   1:L PR[91] 10mm/sec CNT100;
   1:  PR[GP1:91,1] = PR[GP1:90,1] + 6.355;
   1:  PR[GP1:91,2] = PR[GP1:90,2] + -5.589;
   1:L PR[91] 10mm/sec CNT100;
   1:  PR[GP1:91,1] = PR[GP1:90,1] + 7.372;
   1:  PR[GP1:91,2] = PR[GP1:90,2] + -9.674;
   1:L PR[91] 10mm/sec CNT100;
   1:  PR[GP1:91,1] = PR[GP1:90,1] + 8.367;
   1:  PR[GP1:91,2] = PR[GP1:90,2] + -12.675;
   1:L PR[91] 10mm/sec CNT100;
   1:  PR[GP1:91,1] = PR[GP1:90,1] + 10.321;
   1:  PR[GP1:91,2] = PR[GP1:90,2] + -16.925;
   1:L PR[91] 10mm/sec CNT100;
   1:  PR[GP1:91,1] = PR[GP1:90,1] + 13.045;
   1:  PR[GP1:91,2] = PR[GP1:90,2] + -20.757;
   1:L PR[91] 10mm/sec CNT100;
   1:  PR[GP1:91,1] = PR[GP1:90,1] + 14.879;
   1:  PR[GP1:91,2] = PR[GP1:90,2] + -23.159;
   1:L PR[91] 10mm/sec CNT100;
   1:  PR[GP1:91,1] = PR[GP1:90,1] + 18.319;
   1:  PR[GP1:91,2] = PR[GP1:90,2] + -26.468;
   1:L PR[91] 10mm/sec CNT100;
   1:  PR[GP1:91,1] = PR[GP1:90,1] + 22.355;
   1:  PR[GP1:91,2] = PR[GP1:90,2] + -29.107;
   1:L PR[91] 10mm/sec CNT100;
   1:  PR[GP1:91,1] = PR[GP1:90,1] + 24.727;
   1:  PR[GP1:91,2] = PR[GP1:90,2] + -30.680;
   1:L PR[91] 10mm/sec CNT100;
   1:  PR[GP1:91,1] = PR[GP1:90,1] + 29.246;
   1:  PR[GP1:91,2] = PR[GP1:90,2] + -32.548;
   1:L PR[91] 10mm/sec CNT100;
   1:  PR[GP1:91,1] = PR[GP1:90,1] + 34.105;
   1:  PR[GP1:91,2] = PR[GP1:90,2] + -33.559;
   1:L PR[91] 10mm/sec CNT100;
   1:  PR[GP1:91,1] = PR[GP1:90,1] + 36.667;
   1:  PR[GP1:91,2] = PR[GP1:90,2] + -34.223;
   1:L PR[91] 10mm/sec CNT100;
   1:  PR[GP1:91,1] = PR[GP1:90,1] + 41.699;
   1:  PR[GP1:91,2] = PR[GP1:90,2] + -34.315;
   1:L PR[91] 10mm/sec CNT100;
   1:  PR[GP1:91,1] = PR[GP1:90,1] + 44.031;
   1:  PR[GP1:91,2] = PR[GP1:90,2] + -34.139;
   1:L PR[91] 10mm/sec CNT100;
   1:  PR[GP1:91,1] = PR[GP1:90,1] + 49.115;
   1:  PR[GP1:91,2] = PR[GP1:90,2] + -33.273;
   1:L PR[91] 10mm/sec CNT100;
   1:  PR[GP1:91,1] = PR[GP1:90,1] + 53.961;
   1:  PR[GP1:91,2] = PR[GP1:90,2] + -31.473;
   1:L PR[91] 10mm/sec CNT100;
   1:  PR[GP1:91,1] = PR[GP1:90,1] + 55.965;
   1:  PR[GP1:91,2] = PR[GP1:90,2] + -30.610;
   1:L PR[91] 10mm/sec CNT100;
   1:  PR[GP1:91,1] = PR[GP1:90,1] + 60.444;
   1:  PR[GP1:91,2] = PR[GP1:90,2] + -27.909;
   1:L PR[91] 10mm/sec CNT100;
   1:  PR[GP1:91,1] = PR[GP1:90,1] + 64.372;
   1:  PR[GP1:91,2] = PR[GP1:90,2] + -24.396;
   1:L PR[91] 10mm/sec CNT100;
   1:  PR[GP1:91,1] = PR[GP1:90,1] + 65.892;
   1:  PR[GP1:91,2] = PR[GP1:90,2] + -23.011;
   1:L PR[91] 10mm/sec CNT100;
   1:  PR[GP1:91,1] = PR[GP1:90,1] + 69.105;
   1:  PR[GP1:91,2] = PR[GP1:90,2] + -18.822;
   1:L PR[91] 10mm/sec CNT100;
   1:  PR[GP1:91,1] = PR[GP1:90,1] + 71.512;
   1:  PR[GP1:91,2] = PR[GP1:90,2] + -14.052;
   1:L PR[91] 10mm/sec CNT100;
   1:  PR[GP1:91,1] = PR[GP1:90,1] + 72.452;
   1:  PR[GP1:91,2] = PR[GP1:90,2] + -12.328;
   1:L PR[91] 10mm/sec CNT100;
   1:  PR[GP1:91,1] = PR[GP1:90,1] + 73.920;
   1:  PR[GP1:91,2] = PR[GP1:90,2] + -7.231;
   1:L PR[91] 10mm/sec CNT100;
   1:  PR[GP1:91,1] = PR[GP1:90,1] + 74.423;
   1:  PR[GP1:91,2] = PR[GP1:90,2] + -1.863;
   1:L PR[91] 10mm/sec CNT100;
   1:  PR[GP1:91,1] = PR[GP1:90,1] + 74.736;
   1:  PR[GP1:91,2] = PR[GP1:90,2] + 0.017;
   1:L PR[91] 10mm/sec CNT100;
   1:  PR[GP1:91,1] = PR[GP1:90,1] + 74.236;
   1:  PR[GP1:91,2] = PR[GP1:90,2] + 5.360;
   1:L PR[91] 10mm/sec CNT100;
   1:  PR[GP1:91,1] = PR[GP1:90,1] + 73.926;
   1:  PR[GP1:91,2] = PR[GP1:90,2] + 7.201;
   1:L PR[91] 10mm/sec CNT100;
   1:  PR[GP1:91,1] = PR[GP1:90,1] + 72.449;
   1:  PR[GP1:91,2] = PR[GP1:90,2] + 12.328;
   1:L PR[91] 10mm/sec CNT100;
   1:  PR[GP1:91,1] = PR[GP1:90,1] + 70.034;
   1:  PR[GP1:91,2] = PR[GP1:90,2] + 17.114;
   1:L PR[91] 10mm/sec CNT100;
   1:  PR[GP1:91,1] = PR[GP1:90,1] + 69.111;
   1:  PR[GP1:91,2] = PR[GP1:90,2] + 18.805;
   1:L PR[91] 10mm/sec CNT100;
   1:  PR[GP1:91,1] = PR[GP1:90,1] + 65.893;
   1:  PR[GP1:91,2] = PR[GP1:90,2] + 23.000;
   1:L PR[91] 10mm/sec CNT100;
   1:  PR[GP1:91,1] = PR[GP1:90,1] + 61.915;
   1:  PR[GP1:91,2] = PR[GP1:90,2] + 26.557;
   1:L PR[91] 10mm/sec CNT100;
   1:  PR[GP1:91,1] = PR[GP1:90,1] + 60.442;
   1:  PR[GP1:91,2] = PR[GP1:90,2] + 27.901;
   1:L PR[91] 10mm/sec CNT100;
   1:  PR[GP1:91,1] = PR[GP1:90,1] + 55.978;
   1:  PR[GP1:91,2] = PR[GP1:90,2] + 30.593;
   1:L PR[91] 10mm/sec CNT100;
   1:  PR[GP1:91,1] = PR[GP1:90,1] + 51.021;
   1:  PR[GP1:91,2] = PR[GP1:90,2] + 32.434;
   1:L PR[91] 10mm/sec CNT100;
   1:  PR[GP1:91,1] = PR[GP1:90,1] + 49.099;
   1:  PR[GP1:91,2] = PR[GP1:90,2] + 33.267;
   1:L PR[91] 10mm/sec CNT100;
   1:  PR[GP1:91,1] = PR[GP1:90,1] + 44.031;
   1:  PR[GP1:91,2] = PR[GP1:90,2] + 34.130;
   1:L PR[91] 10mm/sec CNT100;
   1:  PR[GP1:91,1] = PR[GP1:90,1] + 41.699;
   1:  PR[GP1:91,2] = PR[GP1:90,2] + 34.306;
   1:L PR[91] 10mm/sec CNT100;
   1:  PR[GP1:91,1] = PR[GP1:90,1] + 36.653;
   1:  PR[GP1:91,2] = PR[GP1:90,2] + 34.214;
   1:L PR[91] 10mm/sec CNT100;
   1:  PR[GP1:91,1] = PR[GP1:90,1] + 31.699;
   1:  PR[GP1:91,2] = PR[GP1:90,2] + 33.183;
   1:L PR[91] 10mm/sec CNT100;
   1:  PR[GP1:91,1] = PR[GP1:90,1] + 29.260;
   1:  PR[GP1:91,2] = PR[GP1:90,2] + 32.545;
   1:L PR[91] 10mm/sec CNT100;
   1:  PR[GP1:91,1] = PR[GP1:90,1] + 24.725;
   1:  PR[GP1:91,2] = PR[GP1:90,2] + 30.670;
   1:L PR[91] 10mm/sec CNT100;
   1:  PR[GP1:91,1] = PR[GP1:90,1] + 20.585;
   1:  PR[GP1:91,2] = PR[GP1:90,2] + 27.963;
   1:L PR[91] 10mm/sec CNT100;
   1:  PR[GP1:91,1] = PR[GP1:90,1] + 18.321;
   1:  PR[GP1:91,2] = PR[GP1:90,2] + 26.461;
   1:L PR[91] 10mm/sec CNT100;
   1:  PR[GP1:91,1] = PR[GP1:90,1] + 14.886;
   1:  PR[GP1:91,2] = PR[GP1:90,2] + 23.157;
   1:L PR[91] 10mm/sec CNT100;
   1:  PR[GP1:91,1] = PR[GP1:90,1] + 12.088;
   1:  PR[GP1:91,2] = PR[GP1:90,2] + 19.220;
   1:L PR[91] 10mm/sec CNT100;
   1:  PR[GP1:91,1] = PR[GP1:90,1] + 10.317;
   1:  PR[GP1:91,2] = PR[GP1:90,2] + 16.907;
   1:L PR[91] 10mm/sec CNT100;
   1:  PR[GP1:91,1] = PR[GP1:90,1] + 8.367;
   1:  PR[GP1:91,2] = PR[GP1:90,2] + 12.666;
   1:L PR[91] 10mm/sec CNT100;
   1:  PR[GP1:91,1] = PR[GP1:90,1] + 7.372;
   1:  PR[GP1:91,2] = PR[GP1:90,2] + 9.665;
   1:L PR[91] 10mm/sec CNT100;
   1:  PR[GP1:91,1] = PR[GP1:90,1] + 6.354;
   1:  PR[GP1:91,2] = PR[GP1:90,2] + 5.577;
   1:L PR[91] 10mm/sec CNT100;
   1:  PR[GP1:91,1] = PR[GP1:90,1] + 6.524;
   1:  PR[GP1:91,2] = PR[GP1:90,2] + 5.479;
   1:L PR[91] 10mm/sec CNT100;
   1:  PR[GP1:91,1] = PR[GP1:90,1] + 5.914;
   1:  PR[GP1:91,2] = PR[GP1:90,2] + 4.305;
   1:L PR[91] 10mm/sec CNT100;
   1:  PR[GP1:91,1] = PR[GP1:90,1] + 4.686;
   1:  PR[GP1:91,2] = PR[GP1:90,2] + 2.087;
   1:L PR[91] 10mm/sec CNT100;
   1:  PR[GP1:91,1] = PR[GP1:90,1] + 4.389;
   1:  PR[GP1:91,2] = PR[GP1:90,2] + 1.764;
   1:L PR[91] 10mm/sec CNT100;
   1:  PR[GP1:91,1] = PR[GP1:90,1] + 3.955;
   1:  PR[GP1:91,2] = PR[GP1:90,2] + 1.465;
   1:L PR[91] 10mm/sec CNT100;
   1:  PR[GP1:91,1] = PR[GP1:90,1] + 1.605;
   1:  PR[GP1:91,2] = PR[GP1:90,2] + 0.594;
   1:L PR[91] 10mm/sec CNT100;
   1:  PR[GP1:91,1] = PR[GP1:90,1] + 0.862;
   1:  PR[GP1:91,2] = PR[GP1:90,2] + 0.396;
   1:L PR[91] 10mm/sec CNT100;
   1:  PR[GP1:91,1] = PR[GP1:90,1] + -0.072;
   1:L PR[91] 10mm/sec CNT100;
   1:  PR[GP1:91,1] = PR[GP1:90,1] + -1.424;
   1:  PR[GP1:91,2] = PR[GP1:90,2] + 0.956;
   1:  PR[GP1:91,3] = PR[GP1:90,3] + 11.970;
   1:L PR[91] 10mm/sec CNT100;
   1:  PR[GP1:91,1] = PR[GP1:90,1] + -1.547;
   1:  PR[GP1:91,2] = PR[GP1:90,2] + 0.962;
   1:L PR[91] 10mm/sec CNT100;
   1:  PR[GP1:91,1] = PR[GP1:90,1] + -3.479;
   1:  PR[GP1:91,2] = PR[GP1:90,2] + 1.726;
   1:L PR[91] 10mm/sec CNT100;
   1:  PR[GP1:91,1] = PR[GP1:90,1] + -4.374;
   1:  PR[GP1:91,2] = PR[GP1:90,2] + 3.341;
   1:L PR[91] 10mm/sec CNT100;
   1:  PR[GP1:91,1] = PR[GP1:90,1] + -4.406;
   1:  PR[GP1:91,2] = PR[GP1:90,2] + 3.371;
   1:L PR[91] 10mm/sec CNT100;
   1:  PR[GP1:91,1] = PR[GP1:90,1] + -5.693;
   1:  PR[GP1:91,2] = PR[GP1:90,2] + 5.463;
   1:L PR[91] 10mm/sec CNT100;
   1:  PR[GP1:91,1] = PR[GP1:90,1] + -5.438;
   1:  PR[GP1:91,2] = PR[GP1:90,2] + 5.607;
   1:L PR[91] 10mm/sec CNT100;
   1:  PR[GP1:91,1] = PR[GP1:90,1] + -6.155;
   1:  PR[GP1:91,2] = PR[GP1:90,2] + 8.483;
   1:L PR[91] 10mm/sec CNT100;
   1:  PR[GP1:91,1] = PR[GP1:90,1] + -7.832;
   1:  PR[GP1:91,2] = PR[GP1:90,2] + 13.544;
   1:L PR[91] 10mm/sec CNT100;
   1:  PR[GP1:91,1] = PR[GP1:90,1] + -9.289;
   1:  PR[GP1:91,2] = PR[GP1:90,2] + 16.715;
   1:L PR[91] 10mm/sec CNT100;
   1:  PR[GP1:91,1] = PR[GP1:90,1] + -11.324;
   1:  PR[GP1:91,2] = PR[GP1:90,2] + 19.577;
   1:L PR[91] 10mm/sec CNT100;
   1:  PR[GP1:91,1] = PR[GP1:90,1] + -14.416;
   1:  PR[GP1:91,2] = PR[GP1:90,2] + 23.625;
   1:L PR[91] 10mm/sec CNT100;
   1:  PR[GP1:91,1] = PR[GP1:90,1] + -17.052;
   1:  PR[GP1:91,2] = PR[GP1:90,2] + 26.160;
   1:L PR[91] 10mm/sec CNT100;
   1:  PR[GP1:91,1] = PR[GP1:90,1] + -20.154;
   1:  PR[GP1:91,2] = PR[GP1:90,2] + 28.188;
   1:L PR[91] 10mm/sec CNT100;
   1:  PR[GP1:91,1] = PR[GP1:90,1] + -24.154;
   1:  PR[GP1:91,2] = PR[GP1:90,2] + 30.842;
   1:L PR[91] 10mm/sec CNT100;
   1:  PR[GP1:91,1] = PR[GP1:90,1] + -27.722;
   1:  PR[GP1:91,2] = PR[GP1:90,2] + 32.317;
   1:L PR[91] 10mm/sec CNT100;
   1:  PR[GP1:91,1] = PR[GP1:90,1] + -31.573;
   1:  PR[GP1:91,2] = PR[GP1:90,2] + 33.118;
   1:L PR[91] 10mm/sec CNT100;
   1:  PR[GP1:91,1] = PR[GP1:90,1] + -35.898;
   1:  PR[GP1:91,2] = PR[GP1:90,2] + 34.238;
   1:L PR[91] 10mm/sec CNT100;
   1:  PR[GP1:91,1] = PR[GP1:90,1] + -39.986;
   1:  PR[GP1:91,2] = PR[GP1:90,2] + 34.312;
   1:L PR[91] 10mm/sec CNT100;
   1:  PR[GP1:91,1] = PR[GP1:90,1] + -43.926;
   1:  PR[GP1:91,2] = PR[GP1:90,2] + 34.016;
   1:L PR[91] 10mm/sec CNT100;
   1:  PR[GP1:91,1] = PR[GP1:90,1] + -48.152;
   1:  PR[GP1:91,2] = PR[GP1:90,2] + 33.296;
   1:L PR[91] 10mm/sec CNT100;
   1:  PR[GP1:91,1] = PR[GP1:90,1] + -52.182;
   1:  PR[GP1:91,2] = PR[GP1:90,2] + 31.799;
   1:L PR[91] 10mm/sec CNT100;
   1:  PR[GP1:91,1] = PR[GP1:90,1] + -55.570;
   1:  PR[GP1:91,2] = PR[GP1:90,2] + 30.339;
   1:L PR[91] 10mm/sec CNT100;
   1:  PR[GP1:91,1] = PR[GP1:90,1] + -59.354;
   1:  PR[GP1:91,2] = PR[GP1:90,2] + 28.057;
   1:L PR[91] 10mm/sec CNT100;
   1:  PR[GP1:91,1] = PR[GP1:90,1] + -62.677;
   1:  PR[GP1:91,2] = PR[GP1:90,2] + 25.086;
   1:L PR[91] 10mm/sec CNT100;
   1:  PR[GP1:91,1] = PR[GP1:90,1] + -65.248;
   1:  PR[GP1:91,2] = PR[GP1:90,2] + 22.743;
   1:L PR[91] 10mm/sec CNT100;
   1:  PR[GP1:91,1] = PR[GP1:90,1] + -67.992;
   1:  PR[GP1:91,2] = PR[GP1:90,2] + 19.165;
   1:L PR[91] 10mm/sec CNT100;
   1:  PR[GP1:91,1] = PR[GP1:90,1] + -70.053;
   1:  PR[GP1:91,2] = PR[GP1:90,2] + 15.082;
   1:L PR[91] 10mm/sec CNT100;
   1:  PR[GP1:91,1] = PR[GP1:90,1] + -71.643;
   1:  PR[GP1:91,2] = PR[GP1:90,2] + 12.163;
   1:L PR[91] 10mm/sec CNT100;
   1:  PR[GP1:91,1] = PR[GP1:90,1] + -72.905;
   1:  PR[GP1:91,2] = PR[GP1:90,2] + 7.782;
   1:L PR[91] 10mm/sec CNT100;
   1:  PR[GP1:91,1] = PR[GP1:90,1] + -73.338;
   1:  PR[GP1:91,2] = PR[GP1:90,2] + 3.156;
   1:L PR[91] 10mm/sec CNT100;
   1:  PR[GP1:91,1] = PR[GP1:90,1] + -73.869;
   1:  PR[GP1:91,2] = PR[GP1:90,2] + -0.026;
   1:L PR[91] 10mm/sec CNT100;
   1:  PR[GP1:91,1] = PR[GP1:90,1] + -73.436;
   1:  PR[GP1:91,2] = PR[GP1:90,2] + -4.653;
   1:L PR[91] 10mm/sec CNT100;
   1:  PR[GP1:91,1] = PR[GP1:90,1] + -72.911;
   1:  PR[GP1:91,2] = PR[GP1:90,2] + -7.770;
   1:L PR[91] 10mm/sec CNT100;
   1:  PR[GP1:91,1] = PR[GP1:90,1] + -71.641;
   1:  PR[GP1:91,2] = PR[GP1:90,2] + -12.181;
   1:L PR[91] 10mm/sec CNT100;
   1:  PR[GP1:91,1] = PR[GP1:90,1] + -69.561;
   1:  PR[GP1:91,2] = PR[GP1:90,2] + -16.301;
   1:L PR[91] 10mm/sec CNT100;
   1:  PR[GP1:91,1] = PR[GP1:90,1] + -67.998;
   1:  PR[GP1:91,2] = PR[GP1:90,2] + -19.166;
   1:L PR[91] 10mm/sec CNT100;
   1:  PR[GP1:91,1] = PR[GP1:90,1] + -65.249;
   1:  PR[GP1:91,2] = PR[GP1:90,2] + -22.750;
   1:L PR[91] 10mm/sec CNT100;
   1:  PR[GP1:91,1] = PR[GP1:90,1] + -61.846;
   1:  PR[GP1:91,2] = PR[GP1:90,2] + -25.794;
   1:L PR[91] 10mm/sec CNT100;
   1:  PR[GP1:91,1] = PR[GP1:90,1] + -59.352;
   1:  PR[GP1:91,2] = PR[GP1:90,2] + -28.067;
   1:L PR[91] 10mm/sec CNT100;
   1:  PR[GP1:91,1] = PR[GP1:90,1] + -55.583;
   1:  PR[GP1:91,2] = PR[GP1:90,2] + -30.340;
   1:L PR[91] 10mm/sec CNT100;
   1:  PR[GP1:91,1] = PR[GP1:90,1] + -51.387;
   1:  PR[GP1:91,2] = PR[GP1:90,2] + -31.899;
   1:L PR[91] 10mm/sec CNT100;
   1:  PR[GP1:91,1] = PR[GP1:90,1] + -48.136;
   1:  PR[GP1:91,2] = PR[GP1:90,2] + -33.307;
   1:L PR[91] 10mm/sec CNT100;
   1:  PR[GP1:91,1] = PR[GP1:90,1] + -43.926;
   1:  PR[GP1:91,2] = PR[GP1:90,2] + -34.025;
   1:L PR[91] 10mm/sec CNT100;
   1:  PR[GP1:91,1] = PR[GP1:90,1] + -39.986;
   1:  PR[GP1:91,2] = PR[GP1:90,2] + -34.321;
   1:L PR[91] 10mm/sec CNT100;
   1:  PR[GP1:91,1] = PR[GP1:90,1] + -35.883;
   1:  PR[GP1:91,2] = PR[GP1:90,2] + -34.247;
   1:L PR[91] 10mm/sec CNT100;
   1:  PR[GP1:91,1] = PR[GP1:90,1] + -31.854;
   1:  PR[GP1:91,2] = PR[GP1:90,2] + -33.408;
   1:L PR[91] 10mm/sec CNT100;
   1:  PR[GP1:91,1] = PR[GP1:90,1] + -27.736;
   1:  PR[GP1:91,2] = PR[GP1:90,2] + -32.331;
   1:L PR[91] 10mm/sec CNT100;
   1:  PR[GP1:91,1] = PR[GP1:90,1] + -24.152;
   1:  PR[GP1:91,2] = PR[GP1:90,2] + -30.850;
   1:L PR[91] 10mm/sec CNT100;
   1:  PR[GP1:91,1] = PR[GP1:90,1] + -20.874;
   1:  PR[GP1:91,2] = PR[GP1:90,2] + -28.706;
   1:L PR[91] 10mm/sec CNT100;
   1:  PR[GP1:91,1] = PR[GP1:90,1] + -17.054;
   1:  PR[GP1:91,2] = PR[GP1:90,2] + -26.171;
   1:L PR[91] 10mm/sec CNT100;
   1:  PR[GP1:91,1] = PR[GP1:90,1] + -14.423;
   1:  PR[GP1:91,2] = PR[GP1:90,2] + -23.641;
   1:L PR[91] 10mm/sec CNT100;
   1:  PR[GP1:91,1] = PR[GP1:90,1] + -12.272;
   1:  PR[GP1:91,2] = PR[GP1:90,2] + -20.613;
   1:L PR[91] 10mm/sec CNT100;
   1:  PR[GP1:91,1] = PR[GP1:90,1] + -9.285;
   1:  PR[GP1:91,2] = PR[GP1:90,2] + -16.713;
   1:L PR[91] 10mm/sec CNT100;
   1:  PR[GP1:91,1] = PR[GP1:90,1] + -7.832;
   1:  PR[GP1:91,2] = PR[GP1:90,2] + -13.553;
   1:L PR[91] 10mm/sec CNT100;
   1:  PR[GP1:91,1] = PR[GP1:90,1] + -6.155;
   1:  PR[GP1:91,2] = PR[GP1:90,2] + -8.493;
   1:L PR[91] 10mm/sec CNT100;
   1:  PR[GP1:91,1] = PR[GP1:90,1] + -5.437;
   1:  PR[GP1:91,2] = PR[GP1:90,2] + -5.610;
   1:L PR[91] 10mm/sec CNT100;
   1:  PR[GP1:91,1] = PR[GP1:90,1] + -5.649;
   1:  PR[GP1:91,2] = PR[GP1:90,2] + -5.486;
   1:L PR[91] 10mm/sec CNT100;
   1:  PR[GP1:91,1] = PR[GP1:90,1] + -4.810;
   1:  PR[GP1:91,2] = PR[GP1:90,2] + -3.871;
   1:L PR[91] 10mm/sec CNT100;
   1:  PR[GP1:91,1] = PR[GP1:90,1] + -3.915;
   1:  PR[GP1:91,2] = PR[GP1:90,2] + -2.254;
   1:L PR[91] 10mm/sec CNT100;
   1:  PR[GP1:91,1] = PR[GP1:90,1] + -3.482;
   1:  PR[GP1:91,2] = PR[GP1:90,2] + -1.784;
   1:L PR[91] 10mm/sec CNT100;
   1:  PR[GP1:91,1] = PR[GP1:90,1] + -2.834;
   1:  PR[GP1:91,2] = PR[GP1:90,2] + -1.337;
   1:L PR[91] 10mm/sec CNT100;
   1:  PR[GP1:91,1] = PR[GP1:90,1] + -1.161;
   1:  PR[GP1:91,2] = PR[GP1:90,2] + -0.717;
   1:L PR[91] 10mm/sec CNT100;
   1:  PR[GP1:91,1] = PR[GP1:90,1] + -0.101;
   1:  PR[GP1:91,2] = PR[GP1:90,2] + -0.435;
   1:L PR[91] 10mm/sec CNT100;
   1:  PR[GP1:91,1] = PR[GP1:90,1] + 0.024;
   1:  PR[GP1:91,2] = PR[GP1:90,2] + -0.404;
   1:L PR[91] 10mm/sec CNT100;
   1:  PR[GP1:91,1] = PR[GP1:90,1] + 0.838;
   1:L PR[91] 10mm/sec CNT100;
   1:  PR[GP1:91,1] = PR[GP1:90,1] + 2.244;
   1:  PR[GP1:91,2] = PR[GP1:90,2] + -0.965;
   1:L PR[91] 10mm/sec CNT100;
   1:  PR[GP1:91,1] = PR[GP1:90,1] + 2.368;
   1:  PR[GP1:91,2] = PR[GP1:90,2] + -0.970;
   1:L PR[91] 10mm/sec CNT100;
   1:  PR[GP1:91,1] = PR[GP1:90,1] + 4.300;
   1:  PR[GP1:91,2] = PR[GP1:90,2] + -1.735;
   1:L PR[91] 10mm/sec CNT100;
   1:  PR[GP1:91,1] = PR[GP1:90,1] + 5.194;
   1:  PR[GP1:91,2] = PR[GP1:90,2] + -3.350;
   1:L PR[91] 10mm/sec CNT100;
   1:  PR[GP1:91,1] = PR[GP1:90,1] + 5.227;
   1:  PR[GP1:91,2] = PR[GP1:90,2] + -3.380;
   1:L PR[91] 10mm/sec CNT100;
   1:  PR[GP1:91,1] = PR[GP1:90,1] + 6.512;
   1:  PR[GP1:91,2] = PR[GP1:90,2] + -5.470;
   1:L PR[91] 10mm/sec CNT100;
   1:  PR[GP1:91,1] = PR[GP1:90,1] + 6.258;
   1:  PR[GP1:91,2] = PR[GP1:90,2] + -5.615;
   1:L PR[91] 10mm/sec CNT100;
   1:  PR[GP1:91,1] = PR[GP1:90,1] + 6.975;
   1:  PR[GP1:91,2] = PR[GP1:90,2] + -8.494;
   1:L PR[91] 10mm/sec CNT100;
   1:  PR[GP1:91,1] = PR[GP1:90,1] + 8.652;
   1:  PR[GP1:91,2] = PR[GP1:90,2] + -13.551;
   1:L PR[91] 10mm/sec CNT100;
   1:  PR[GP1:91,1] = PR[GP1:90,1] + 10.109;
   1:  PR[GP1:91,2] = PR[GP1:90,2] + -16.721;
   1:L PR[91] 10mm/sec CNT100;
   1:  PR[GP1:91,1] = PR[GP1:90,1] + 12.144;
   1:  PR[GP1:91,2] = PR[GP1:90,2] + -19.584;
   1:L PR[91] 10mm/sec CNT100;
   1:  PR[GP1:91,1] = PR[GP1:90,1] + 15.236;
   1:  PR[GP1:91,2] = PR[GP1:90,2] + -23.633;
   1:L PR[91] 10mm/sec CNT100;
   1:  PR[GP1:91,1] = PR[GP1:90,1] + 17.872;
   1:  PR[GP1:91,2] = PR[GP1:90,2] + -26.169;
   1:L PR[91] 10mm/sec CNT100;
   1:  PR[GP1:91,1] = PR[GP1:90,1] + 20.974;
   1:  PR[GP1:91,2] = PR[GP1:90,2] + -28.196;
   1:L PR[91] 10mm/sec CNT100;
   1:  PR[GP1:91,1] = PR[GP1:90,1] + 24.974;
   1:  PR[GP1:91,2] = PR[GP1:90,2] + -30.850;
   1:L PR[91] 10mm/sec CNT100;
   1:  PR[GP1:91,1] = PR[GP1:90,1] + 28.542;
   1:  PR[GP1:91,2] = PR[GP1:90,2] + -32.325;
   1:L PR[91] 10mm/sec CNT100;
   1:  PR[GP1:91,1] = PR[GP1:90,1] + 32.393;
   1:  PR[GP1:91,2] = PR[GP1:90,2] + -33.126;
   1:L PR[91] 10mm/sec CNT100;
   1:  PR[GP1:91,1] = PR[GP1:90,1] + 36.718;
   1:  PR[GP1:91,2] = PR[GP1:90,2] + -34.247;
   1:L PR[91] 10mm/sec CNT100;
   1:  PR[GP1:91,1] = PR[GP1:90,1] + 40.805;
   1:  PR[GP1:91,2] = PR[GP1:90,2] + -34.321;
   1:L PR[91] 10mm/sec CNT100;
   1:  PR[GP1:91,1] = PR[GP1:90,1] + 44.746;
   1:  PR[GP1:91,2] = PR[GP1:90,2] + -34.025;
   1:L PR[91] 10mm/sec CNT100;
   1:  PR[GP1:91,1] = PR[GP1:90,1] + 48.972;
   1:  PR[GP1:91,2] = PR[GP1:90,2] + -33.305;
   1:L PR[91] 10mm/sec CNT100;
   1:  PR[GP1:91,1] = PR[GP1:90,1] + 53.002;
   1:  PR[GP1:91,2] = PR[GP1:90,2] + -31.807;
   1:L PR[91] 10mm/sec CNT100;
   1:  PR[GP1:91,1] = PR[GP1:90,1] + 56.390;
   1:  PR[GP1:91,2] = PR[GP1:90,2] + -30.348;
   1:L PR[91] 10mm/sec CNT100;
   1:  PR[GP1:91,1] = PR[GP1:90,1] + 60.174;
   1:  PR[GP1:91,2] = PR[GP1:90,2] + -28.066;
   1:L PR[91] 10mm/sec CNT100;
   1:  PR[GP1:91,1] = PR[GP1:90,1] + 63.498;
   1:  PR[GP1:91,2] = PR[GP1:90,2] + -25.095;
   1:L PR[91] 10mm/sec CNT100;
   1:  PR[GP1:91,1] = PR[GP1:90,1] + 66.068;
   1:  PR[GP1:91,2] = PR[GP1:90,2] + -22.752;
   1:L PR[91] 10mm/sec CNT100;
   1:  PR[GP1:91,1] = PR[GP1:90,1] + 68.813;
   1:  PR[GP1:91,2] = PR[GP1:90,2] + -19.173;
   1:L PR[91] 10mm/sec CNT100;
   1:  PR[GP1:91,1] = PR[GP1:90,1] + 70.873;
   1:  PR[GP1:91,2] = PR[GP1:90,2] + -15.091;
   1:L PR[91] 10mm/sec CNT100;
   1:  PR[GP1:91,1] = PR[GP1:90,1] + 72.464;
   1:  PR[GP1:91,2] = PR[GP1:90,2] + -12.173;
   1:L PR[91] 10mm/sec CNT100;
   1:  PR[GP1:91,1] = PR[GP1:90,1] + 73.725;
   1:  PR[GP1:91,2] = PR[GP1:90,2] + -7.792;
   1:L PR[91] 10mm/sec CNT100;
   1:  PR[GP1:91,1] = PR[GP1:90,1] + 74.159;
   1:  PR[GP1:91,2] = PR[GP1:90,2] + -3.166;
   1:L PR[91] 10mm/sec CNT100;
   1:  PR[GP1:91,1] = PR[GP1:90,1] + 74.690;
   1:  PR[GP1:91,2] = PR[GP1:90,2] + 0.017;
   1:L PR[91] 10mm/sec CNT100;
   1:  PR[GP1:91,1] = PR[GP1:90,1] + 74.256;
   1:  PR[GP1:91,2] = PR[GP1:90,2] + 4.644;
   1:L PR[91] 10mm/sec CNT100;
   1:  PR[GP1:91,1] = PR[GP1:90,1] + 73.731;
   1:  PR[GP1:91,2] = PR[GP1:90,2] + 7.762;
   1:L PR[91] 10mm/sec CNT100;
   1:  PR[GP1:91,1] = PR[GP1:90,1] + 72.461;
   1:  PR[GP1:91,2] = PR[GP1:90,2] + 12.173;
   1:L PR[91] 10mm/sec CNT100;
   1:  PR[GP1:91,1] = PR[GP1:90,1] + 70.382;
   1:  PR[GP1:91,2] = PR[GP1:90,2] + 16.293;
   1:L PR[91] 10mm/sec CNT100;
   1:  PR[GP1:91,1] = PR[GP1:90,1] + 68.819;
   1:  PR[GP1:91,2] = PR[GP1:90,2] + 19.157;
   1:L PR[91] 10mm/sec CNT100;
   1:  PR[GP1:91,1] = PR[GP1:90,1] + 66.070;
   1:  PR[GP1:91,2] = PR[GP1:90,2] + 22.741;
   1:L PR[91] 10mm/sec CNT100;
   1:  PR[GP1:91,1] = PR[GP1:90,1] + 62.666;
   1:  PR[GP1:91,2] = PR[GP1:90,2] + 25.784;
   1:L PR[91] 10mm/sec CNT100;
   1:  PR[GP1:91,1] = PR[GP1:90,1] + 60.172;
   1:  PR[GP1:91,2] = PR[GP1:90,2] + 28.059;
   1:L PR[91] 10mm/sec CNT100;
   1:  PR[GP1:91,1] = PR[GP1:90,1] + 56.403;
   1:  PR[GP1:91,2] = PR[GP1:90,2] + 30.332;
   1:L PR[91] 10mm/sec CNT100;
   1:  PR[GP1:91,1] = PR[GP1:90,1] + 52.207;
   1:  PR[GP1:91,2] = PR[GP1:90,2] + 31.890;
   1:L PR[91] 10mm/sec CNT100;
   1:  PR[GP1:91,1] = PR[GP1:90,1] + 48.956;
   1:  PR[GP1:91,2] = PR[GP1:90,2] + 33.298;
   1:L PR[91] 10mm/sec CNT100;
   1:  PR[GP1:91,1] = PR[GP1:90,1] + 44.746;
   1:  PR[GP1:91,2] = PR[GP1:90,2] + 34.016;
   1:L PR[91] 10mm/sec CNT100;
   1:  PR[GP1:91,1] = PR[GP1:90,1] + 40.805;
   1:  PR[GP1:91,2] = PR[GP1:90,2] + 34.312;
   1:L PR[91] 10mm/sec CNT100;
   1:  PR[GP1:91,1] = PR[GP1:90,1] + 36.703;
   1:  PR[GP1:91,2] = PR[GP1:90,2] + 34.238;
   1:L PR[91] 10mm/sec CNT100;
   1:  PR[GP1:91,1] = PR[GP1:90,1] + 32.674;
   1:  PR[GP1:91,2] = PR[GP1:90,2] + 33.399;
   1:L PR[91] 10mm/sec CNT100;
   1:  PR[GP1:91,1] = PR[GP1:90,1] + 28.556;
   1:  PR[GP1:91,2] = PR[GP1:90,2] + 32.322;
   1:L PR[91] 10mm/sec CNT100;
   1:  PR[GP1:91,1] = PR[GP1:90,1] + 24.972;
   1:  PR[GP1:91,2] = PR[GP1:90,2] + 30.840;
   1:L PR[91] 10mm/sec CNT100;
   1:  PR[GP1:91,1] = PR[GP1:90,1] + 21.693;
   1:  PR[GP1:91,2] = PR[GP1:90,2] + 28.696;
   1:L PR[91] 10mm/sec CNT100;
   1:  PR[GP1:91,1] = PR[GP1:90,1] + 17.874;
   1:  PR[GP1:91,2] = PR[GP1:90,2] + 26.161;
   1:L PR[91] 10mm/sec CNT100;
   1:  PR[GP1:91,1] = PR[GP1:90,1] + 15.243;
   1:  PR[GP1:91,2] = PR[GP1:90,2] + 23.631;
   1:L PR[91] 10mm/sec CNT100;
   1:  PR[GP1:91,1] = PR[GP1:90,1] + 13.091;
   1:  PR[GP1:91,2] = PR[GP1:90,2] + 20.604;
   1:L PR[91] 10mm/sec CNT100;
   1:  PR[GP1:91,1] = PR[GP1:90,1] + 10.105;
   1:  PR[GP1:91,2] = PR[GP1:90,2] + 16.703;
   1:L PR[91] 10mm/sec CNT100;
   1:  PR[GP1:91,1] = PR[GP1:90,1] + 8.652;
   1:  PR[GP1:91,2] = PR[GP1:90,2] + 13.542;
   1:L PR[91] 10mm/sec CNT100;
   1:  PR[GP1:91,1] = PR[GP1:90,1] + 6.975;
   1:  PR[GP1:91,2] = PR[GP1:90,2] + 8.484;
   1:L PR[91] 10mm/sec CNT100;
   1:  PR[GP1:91,1] = PR[GP1:90,1] + 6.258;
   1:  PR[GP1:91,2] = PR[GP1:90,2] + 5.602;
   1:L PR[91] 10mm/sec CNT100;
   1:  PR[GP1:91,1] = PR[GP1:90,1] + 6.470;
   1:  PR[GP1:91,2] = PR[GP1:90,2] + 5.479;
   1:L PR[91] 10mm/sec CNT100;
   1:  PR[GP1:91,1] = PR[GP1:90,1] + 5.631;
   1:  PR[GP1:91,2] = PR[GP1:90,2] + 3.863;
   1:L PR[91] 10mm/sec CNT100;
   1:  PR[GP1:91,1] = PR[GP1:90,1] + 4.735;
   1:  PR[GP1:91,2] = PR[GP1:90,2] + 2.246;
   1:L PR[91] 10mm/sec CNT100;
   1:  PR[GP1:91,1] = PR[GP1:90,1] + 4.302;
   1:  PR[GP1:91,2] = PR[GP1:90,2] + 1.775;
   1:L PR[91] 10mm/sec CNT100;
   1:  PR[GP1:91,1] = PR[GP1:90,1] + 3.654;
   1:  PR[GP1:91,2] = PR[GP1:90,2] + 1.329;
   1:L PR[91] 10mm/sec CNT100;
   1:  PR[GP1:91,1] = PR[GP1:90,1] + 1.982;
   1:  PR[GP1:91,2] = PR[GP1:90,2] + 0.708;
   1:L PR[91] 10mm/sec CNT100;
   1:  PR[GP1:91,1] = PR[GP1:90,1] + 0.919;
   1:  PR[GP1:91,2] = PR[GP1:90,2] + 0.425;
   1:L PR[91] 10mm/sec CNT100;
   1:  PR[GP1:91,1] = PR[GP1:90,1] + 0.796;
   1:  PR[GP1:91,2] = PR[GP1:90,2] + 0.396;
   1:L PR[91] 10mm/sec CNT100;
   1:  PR[GP1:91,1] = PR[GP1:90,1] + -0.018;
   1:L PR[91] 10mm/sec CNT100;
   1:  PR[GP1:91,1] = PR[GP1:90,1] + -0.616;
   1:  PR[GP1:91,2] = PR[GP1:90,2] + 0.693;
   1:  PR[GP1:91,3] = PR[GP1:90,3] + 13.300;
   1:L PR[91] 10mm/sec CNT100;
   1:  PR[GP1:91,1] = PR[GP1:90,1] + -0.790;
   1:  PR[GP1:91,2] = PR[GP1:90,2] + 0.701;
   1:L PR[91] 10mm/sec CNT100;
   1:  PR[GP1:91,1] = PR[GP1:90,1] + -3.381;
   1:  PR[GP1:91,2] = PR[GP1:90,2] + 1.726;
   1:L PR[91] 10mm/sec CNT100;
   1:  PR[GP1:91,1] = PR[GP1:90,1] + -3.935;
   1:  PR[GP1:91,2] = PR[GP1:90,2] + 2.726;
   1:L PR[91] 10mm/sec CNT100;
   1:  PR[GP1:91,1] = PR[GP1:90,1] + -3.985;
   1:  PR[GP1:91,2] = PR[GP1:90,2] + 2.772;
   1:L PR[91] 10mm/sec CNT100;
   1:  PR[GP1:91,1] = PR[GP1:90,1] + -4.673;
   1:  PR[GP1:91,2] = PR[GP1:90,2] + 3.890;
   1:L PR[91] 10mm/sec CNT100;
   1:  PR[GP1:91,1] = PR[GP1:90,1] + -5.310;
   1:  PR[GP1:91,2] = PR[GP1:90,2] + 5.066;
   1:L PR[91] 10mm/sec CNT100;
   1:  PR[GP1:91,1] = PR[GP1:90,1] + -5.369;
   1:  PR[GP1:91,2] = PR[GP1:90,2] + 5.616;
   1:L PR[91] 10mm/sec CNT100;
   1:  PR[GP1:91,1] = PR[GP1:90,1] + -5.342;
   1:  PR[GP1:91,2] = PR[GP1:90,2] + 5.632;
   1:L PR[91] 10mm/sec CNT100;
   1:  PR[GP1:91,1] = PR[GP1:90,1] + -5.758;
   1:  PR[GP1:91,2] = PR[GP1:90,2] + 7.303;
   1:L PR[91] 10mm/sec CNT100;
   1:  PR[GP1:91,1] = PR[GP1:90,1] + -8.117;
   1:  PR[GP1:91,2] = PR[GP1:90,2] + 14.421;
   1:L PR[91] 10mm/sec CNT100;
   1:  PR[GP1:91,1] = PR[GP1:90,1] + -9.078;
   1:  PR[GP1:91,2] = PR[GP1:90,2] + 16.511;
   1:L PR[91] 10mm/sec CNT100;
   1:  PR[GP1:91,1] = PR[GP1:90,1] + -10.424;
   1:  PR[GP1:91,2] = PR[GP1:90,2] + 18.405;
   1:L PR[91] 10mm/sec CNT100;
   1:  PR[GP1:91,1] = PR[GP1:90,1] + -14.774;
   1:  PR[GP1:91,2] = PR[GP1:90,2] + 24.099;
   1:L PR[91] 10mm/sec CNT100;
   1:  PR[GP1:91,1] = PR[GP1:90,1] + -16.606;
   1:  PR[GP1:91,2] = PR[GP1:90,2] + 25.861;
   1:L PR[91] 10mm/sec CNT100;
   1:  PR[GP1:91,1] = PR[GP1:90,1] + -18.773;
   1:  PR[GP1:91,2] = PR[GP1:90,2] + 27.278;
   1:L PR[91] 10mm/sec CNT100;
   1:  PR[GP1:91,1] = PR[GP1:90,1] + -24.402;
   1:  PR[GP1:91,2] = PR[GP1:90,2] + 31.012;
   1:L PR[91] 10mm/sec CNT100;
   1:  PR[GP1:91,1] = PR[GP1:90,1] + -27.019;
   1:  PR[GP1:91,2] = PR[GP1:90,2] + 32.094;
   1:L PR[91] 10mm/sec CNT100;
   1:  PR[GP1:91,1] = PR[GP1:90,1] + -29.862;
   1:  PR[GP1:91,2] = PR[GP1:90,2] + 32.685;
   1:L PR[91] 10mm/sec CNT100;
   1:  PR[GP1:91,1] = PR[GP1:90,1] + -35.949;
   1:  PR[GP1:91,2] = PR[GP1:90,2] + 34.262;
   1:L PR[91] 10mm/sec CNT100;
   1:  PR[GP1:91,1] = PR[GP1:90,1] + -39.092;
   1:  PR[GP1:91,2] = PR[GP1:90,2] + 34.319;
   1:L PR[91] 10mm/sec CNT100;
   1:  PR[GP1:91,1] = PR[GP1:90,1] + -44.641;
   1:  PR[GP1:91,2] = PR[GP1:90,2] + 33.901;
   1:L PR[91] 10mm/sec CNT100;
   1:  PR[GP1:91,1] = PR[GP1:90,1] + -48.009;
   1:  PR[GP1:91,2] = PR[GP1:90,2] + 33.327;
   1:L PR[91] 10mm/sec CNT100;
   1:  PR[GP1:91,1] = PR[GP1:90,1] + -51.223;
   1:  PR[GP1:91,2] = PR[GP1:90,2] + 32.133;
   1:L PR[91] 10mm/sec CNT100;
   1:  PR[GP1:91,1] = PR[GP1:90,1] + -55.995;
   1:  PR[GP1:91,2] = PR[GP1:90,2] + 30.078;
   1:L PR[91] 10mm/sec CNT100;
   1:  PR[GP1:91,1] = PR[GP1:90,1] + -59.085;
   1:  PR[GP1:91,2] = PR[GP1:90,2] + 28.215;
   1:L PR[91] 10mm/sec CNT100;
   1:  PR[GP1:91,1] = PR[GP1:90,1] + -61.802;
   1:  PR[GP1:91,2] = PR[GP1:90,2] + 25.785;
   1:L PR[91] 10mm/sec CNT100;
   1:  PR[GP1:91,1] = PR[GP1:90,1] + -65.424;
   1:  PR[GP1:91,2] = PR[GP1:90,2] + 22.484;
   1:L PR[91] 10mm/sec CNT100;
   1:  PR[GP1:91,1] = PR[GP1:90,1] + -67.700;
   1:  PR[GP1:91,2] = PR[GP1:90,2] + 19.516;
   1:L PR[91] 10mm/sec CNT100;
   1:  PR[GP1:91,1] = PR[GP1:90,1] + -69.414;
   1:  PR[GP1:91,2] = PR[GP1:90,2] + 16.122;
   1:L PR[91] 10mm/sec CNT100;
   1:  PR[GP1:91,1] = PR[GP1:90,1] + -71.655;
   1:  PR[GP1:91,2] = PR[GP1:90,2] + 12.007;
   1:L PR[91] 10mm/sec CNT100;
   1:  PR[GP1:91,1] = PR[GP1:90,1] + -72.710;
   1:  PR[GP1:91,2] = PR[GP1:90,2] + 8.343;
   1:L PR[91] 10mm/sec CNT100;
   1:  PR[GP1:91,1] = PR[GP1:90,1] + -73.074;
   1:  PR[GP1:91,2] = PR[GP1:90,2] + 4.459;
   1:L PR[91] 10mm/sec CNT100;
   1:  PR[GP1:91,1] = PR[GP1:90,1] + -73.823;
   1:  PR[GP1:91,2] = PR[GP1:90,2] + -0.026;
   1:L PR[91] 10mm/sec CNT100;
   1:  PR[GP1:91,1] = PR[GP1:90,1] + -73.456;
   1:  PR[GP1:91,2] = PR[GP1:90,2] + -3.937;
   1:L PR[91] 10mm/sec CNT100;
   1:  PR[GP1:91,1] = PR[GP1:90,1] + -72.717;
   1:  PR[GP1:91,2] = PR[GP1:90,2] + -8.330;
   1:L PR[91] 10mm/sec CNT100;
   1:  PR[GP1:91,1] = PR[GP1:90,1] + -71.652;
   1:  PR[GP1:91,2] = PR[GP1:90,2] + -12.025;
   1:L PR[91] 10mm/sec CNT100;
   1:  PR[GP1:91,1] = PR[GP1:90,1] + -69.909;
   1:  PR[GP1:91,2] = PR[GP1:90,2] + -15.479;
   1:L PR[91] 10mm/sec CNT100;
   1:  PR[GP1:91,1] = PR[GP1:90,1] + -67.706;
   1:  PR[GP1:91,2] = PR[GP1:90,2] + -19.518;
   1:L PR[91] 10mm/sec CNT100;
   1:  PR[GP1:91,1] = PR[GP1:90,1] + -65.426;
   1:  PR[GP1:91,2] = PR[GP1:90,2] + -22.491;
   1:L PR[91] 10mm/sec CNT100;
   1:  PR[GP1:91,1] = PR[GP1:90,1] + -62.596;
   1:  PR[GP1:91,2] = PR[GP1:90,2] + -25.021;
   1:L PR[91] 10mm/sec CNT100;
   1:  PR[GP1:91,1] = PR[GP1:90,1] + -59.082;
   1:  PR[GP1:91,2] = PR[GP1:90,2] + -28.225;
   1:L PR[91] 10mm/sec CNT100;
   1:  PR[GP1:91,1] = PR[GP1:90,1] + -56.008;
   1:  PR[GP1:91,2] = PR[GP1:90,2] + -30.078;
   1:L PR[91] 10mm/sec CNT100;
   1:  PR[GP1:91,1] = PR[GP1:90,1] + -52.573;
   1:  PR[GP1:91,2] = PR[GP1:90,2] + -31.354;
   1:L PR[91] 10mm/sec CNT100;
   1:  PR[GP1:91,1] = PR[GP1:90,1] + -47.993;
   1:  PR[GP1:91,2] = PR[GP1:90,2] + -33.339;
   1:L PR[91] 10mm/sec CNT100;
   1:  PR[GP1:91,1] = PR[GP1:90,1] + -44.641;
   1:  PR[GP1:91,2] = PR[GP1:90,2] + -33.910;
   1:L PR[91] 10mm/sec CNT100;
   1:  PR[GP1:91,1] = PR[GP1:90,1] + -39.092;
   1:  PR[GP1:91,2] = PR[GP1:90,2] + -34.328;
   1:L PR[91] 10mm/sec CNT100;
   1:  PR[GP1:91,1] = PR[GP1:90,1] + -35.934;
   1:  PR[GP1:91,2] = PR[GP1:90,2] + -34.270;
   1:L PR[91] 10mm/sec CNT100;
   1:  PR[GP1:91,1] = PR[GP1:90,1] + -32.829;
   1:  PR[GP1:91,2] = PR[GP1:90,2] + -33.624;
   1:L PR[91] 10mm/sec CNT100;
   1:  PR[GP1:91,1] = PR[GP1:90,1] + -27.033;
   1:  PR[GP1:91,2] = PR[GP1:90,2] + -32.108;
   1:L PR[91] 10mm/sec CNT100;
   1:  PR[GP1:91,1] = PR[GP1:90,1] + -24.400;
   1:  PR[GP1:91,2] = PR[GP1:90,2] + -31.020;
   1:L PR[91] 10mm/sec CNT100;
   1:  PR[GP1:91,1] = PR[GP1:90,1] + -21.983;
   1:  PR[GP1:91,2] = PR[GP1:90,2] + -29.440;
   1:L PR[91] 10mm/sec CNT100;
   1:  PR[GP1:91,1] = PR[GP1:90,1] + -16.607;
   1:  PR[GP1:91,2] = PR[GP1:90,2] + -25.872;
   1:L PR[91] 10mm/sec CNT100;
   1:  PR[GP1:91,1] = PR[GP1:90,1] + -14.781;
   1:  PR[GP1:91,2] = PR[GP1:90,2] + -24.115;
   1:L PR[91] 10mm/sec CNT100;
   1:  PR[GP1:91,1] = PR[GP1:90,1] + -13.276;
   1:  PR[GP1:91,2] = PR[GP1:90,2] + -21.997;
   1:L PR[91] 10mm/sec CNT100;
   1:  PR[GP1:91,1] = PR[GP1:90,1] + -9.073;
   1:  PR[GP1:91,2] = PR[GP1:90,2] + -16.510;
   1:L PR[91] 10mm/sec CNT100;
   1:  PR[GP1:91,1] = PR[GP1:90,1] + -8.117;
   1:  PR[GP1:91,2] = PR[GP1:90,2] + -14.430;
   1:L PR[91] 10mm/sec CNT100;
   1:  PR[GP1:91,1] = PR[GP1:90,1] + -5.758;
   1:  PR[GP1:91,2] = PR[GP1:90,2] + -7.313;
   1:L PR[91] 10mm/sec CNT100;
   1:  PR[GP1:91,1] = PR[GP1:90,1] + -5.340;
   1:  PR[GP1:91,2] = PR[GP1:90,2] + -5.635;
   1:L PR[91] 10mm/sec CNT100;
   1:  PR[GP1:91,1] = PR[GP1:90,1] + -5.371;
   1:  PR[GP1:91,2] = PR[GP1:90,2] + -5.618;
   1:L PR[91] 10mm/sec CNT100;
   1:  PR[GP1:91,1] = PR[GP1:90,1] + -5.314;
   1:  PR[GP1:91,2] = PR[GP1:90,2] + -5.104;
   1:L PR[91] 10mm/sec CNT100;
   1:  PR[GP1:91,1] = PR[GP1:90,1] + -4.965;
   1:  PR[GP1:91,2] = PR[GP1:90,2] + -4.273;
   1:L PR[91] 10mm/sec CNT100;
   1:  PR[GP1:91,1] = PR[GP1:90,1] + -4.526;
   1:  PR[GP1:91,2] = PR[GP1:90,2] + -3.429;
   1:L PR[91] 10mm/sec CNT100;
   1:  PR[GP1:91,1] = PR[GP1:90,1] + -3.964;
   1:  PR[GP1:91,2] = PR[GP1:90,2] + -2.413;
   1:L PR[91] 10mm/sec CNT100;
   1:  PR[GP1:91,1] = PR[GP1:90,1] + -3.395;
   1:  PR[GP1:91,2] = PR[GP1:90,2] + -1.795;
   1:L PR[91] 10mm/sec CNT100;
   1:  PR[GP1:91,1] = PR[GP1:90,1] + -2.533;
   1:  PR[GP1:91,2] = PR[GP1:90,2] + -1.201;
   1:L PR[91] 10mm/sec CNT100;
   1:  PR[GP1:91,1] = PR[GP1:90,1] + -1.538;
   1:  PR[GP1:91,2] = PR[GP1:90,2] + -0.832;
   1:L PR[91] 10mm/sec CNT100;
   1:  PR[GP1:91,1] = PR[GP1:90,1] + -0.919;
   1:  PR[GP1:91,2] = PR[GP1:90,2] + -0.667;
   1:L PR[91] 10mm/sec CNT100;
   1:  PR[GP1:91,1] = PR[GP1:90,1] + 0.173;
   1:  PR[GP1:91,2] = PR[GP1:90,2] + -0.404;
   1:L PR[91] 10mm/sec CNT100;
   1:  PR[GP1:91,1] = PR[GP1:90,1] + 0.690;
   1:L PR[91] 10mm/sec CNT100;
   1:  PR[GP1:91,1] = PR[GP1:90,1] + 1.437;
   1:  PR[GP1:91,2] = PR[GP1:90,2] + -0.702;
   1:L PR[91] 10mm/sec CNT100;
   1:  PR[GP1:91,1] = PR[GP1:90,1] + 1.611;
   1:  PR[GP1:91,2] = PR[GP1:90,2] + -0.710;
   1:L PR[91] 10mm/sec CNT100;
   1:  PR[GP1:91,1] = PR[GP1:90,1] + 4.202;
   1:  PR[GP1:91,2] = PR[GP1:90,2] + -1.735;
   1:L PR[91] 10mm/sec CNT100;
   1:  PR[GP1:91,1] = PR[GP1:90,1] + 4.756;
   1:  PR[GP1:91,2] = PR[GP1:90,2] + -2.736;
   1:L PR[91] 10mm/sec CNT100;
   1:  PR[GP1:91,1] = PR[GP1:90,1] + 4.806;
   1:  PR[GP1:91,2] = PR[GP1:90,2] + -2.781;
   1:L PR[91] 10mm/sec CNT100;
   1:  PR[GP1:91,1] = PR[GP1:90,1] + 5.494;
   1:  PR[GP1:91,2] = PR[GP1:90,2] + -3.900;
   1:L PR[91] 10mm/sec CNT100;
   1:  PR[GP1:91,1] = PR[GP1:90,1] + 6.130;
   1:  PR[GP1:91,2] = PR[GP1:90,2] + -5.075;
   1:L PR[91] 10mm/sec CNT100;
   1:  PR[GP1:91,1] = PR[GP1:90,1] + 6.190;
   1:  PR[GP1:91,2] = PR[GP1:90,2] + -5.625;
   1:L PR[91] 10mm/sec CNT100;
   1:  PR[GP1:91,1] = PR[GP1:90,1] + 6.162;
   1:  PR[GP1:91,2] = PR[GP1:90,2] + -5.640;
   1:L PR[91] 10mm/sec CNT100;
   1:  PR[GP1:91,1] = PR[GP1:90,1] + 6.578;
   1:  PR[GP1:91,2] = PR[GP1:90,2] + -7.314;
   1:L PR[91] 10mm/sec CNT100;
   1:  PR[GP1:91,1] = PR[GP1:90,1] + 8.936;
   1:  PR[GP1:91,2] = PR[GP1:90,2] + -14.427;
   1:L PR[91] 10mm/sec CNT100;
   1:  PR[GP1:91,1] = PR[GP1:90,1] + 9.897;
   1:  PR[GP1:91,2] = PR[GP1:90,2] + -16.517;
   1:L PR[91] 10mm/sec CNT100;
   1:  PR[GP1:91,1] = PR[GP1:90,1] + 11.243;
   1:  PR[GP1:91,2] = PR[GP1:90,2] + -18.411;
   1:L PR[91] 10mm/sec CNT100;
   1:  PR[GP1:91,1] = PR[GP1:90,1] + 15.593;
   1:  PR[GP1:91,2] = PR[GP1:90,2] + -24.107;
   1:L PR[91] 10mm/sec CNT100;
   1:  PR[GP1:91,1] = PR[GP1:90,1] + 17.425;
   1:  PR[GP1:91,2] = PR[GP1:90,2] + -25.869;
   1:L PR[91] 10mm/sec CNT100;
   1:  PR[GP1:91,1] = PR[GP1:90,1] + 19.593;
   1:  PR[GP1:91,2] = PR[GP1:90,2] + -27.286;
   1:L PR[91] 10mm/sec CNT100;
   1:  PR[GP1:91,1] = PR[GP1:90,1] + 25.221;
   1:  PR[GP1:91,2] = PR[GP1:90,2] + -31.020;
   1:L PR[91] 10mm/sec CNT100;
   1:  PR[GP1:91,1] = PR[GP1:90,1] + 27.838;
   1:  PR[GP1:91,2] = PR[GP1:90,2] + -32.102;
   1:L PR[91] 10mm/sec CNT100;
   1:  PR[GP1:91,1] = PR[GP1:90,1] + 30.681;
   1:  PR[GP1:91,2] = PR[GP1:90,2] + -32.694;
   1:L PR[91] 10mm/sec CNT100;
   1:  PR[GP1:91,1] = PR[GP1:90,1] + 36.769;
   1:  PR[GP1:91,2] = PR[GP1:90,2] + -34.270;
   1:L PR[91] 10mm/sec CNT100;
   1:  PR[GP1:91,1] = PR[GP1:90,1] + 39.912;
   1:  PR[GP1:91,2] = PR[GP1:90,2] + -34.328;
   1:L PR[91] 10mm/sec CNT100;
   1:  PR[GP1:91,1] = PR[GP1:90,1] + 45.461;
   1:  PR[GP1:91,2] = PR[GP1:90,2] + -33.910;
   1:L PR[91] 10mm/sec CNT100;
   1:  PR[GP1:91,1] = PR[GP1:90,1] + 48.829;
   1:  PR[GP1:91,2] = PR[GP1:90,2] + -33.336;
   1:L PR[91] 10mm/sec CNT100;
   1:  PR[GP1:91,1] = PR[GP1:90,1] + 52.043;
   1:  PR[GP1:91,2] = PR[GP1:90,2] + -32.142;
   1:L PR[91] 10mm/sec CNT100;
   1:  PR[GP1:91,1] = PR[GP1:90,1] + 56.816;
   1:  PR[GP1:91,2] = PR[GP1:90,2] + -30.087;
   1:L PR[91] 10mm/sec CNT100;
   1:  PR[GP1:91,1] = PR[GP1:90,1] + 59.905;
   1:  PR[GP1:91,2] = PR[GP1:90,2] + -28.224;
   1:L PR[91] 10mm/sec CNT100;
   1:  PR[GP1:91,1] = PR[GP1:90,1] + 62.623;
   1:  PR[GP1:91,2] = PR[GP1:90,2] + -25.794;
   1:L PR[91] 10mm/sec CNT100;
   1:  PR[GP1:91,1] = PR[GP1:90,1] + 66.245;
   1:  PR[GP1:91,2] = PR[GP1:90,2] + -22.492;
   1:L PR[91] 10mm/sec CNT100;
   1:  PR[GP1:91,1] = PR[GP1:90,1] + 68.521;
   1:  PR[GP1:91,2] = PR[GP1:90,2] + -19.525;
   1:L PR[91] 10mm/sec CNT100;
   1:  PR[GP1:91,1] = PR[GP1:90,1] + 70.234;
   1:  PR[GP1:91,2] = PR[GP1:90,2] + -16.130;
   1:L PR[91] 10mm/sec CNT100;
   1:  PR[GP1:91,1] = PR[GP1:90,1] + 72.476;
   1:  PR[GP1:91,2] = PR[GP1:90,2] + -12.018;
   1:L PR[91] 10mm/sec CNT100;
   1:  PR[GP1:91,1] = PR[GP1:90,1] + 73.531;
   1:  PR[GP1:91,2] = PR[GP1:90,2] + -8.354;
   1:L PR[91] 10mm/sec CNT100;
   1:  PR[GP1:91,1] = PR[GP1:90,1] + 73.895;
   1:  PR[GP1:91,2] = PR[GP1:90,2] + -4.470;
   1:L PR[91] 10mm/sec CNT100;
   1:  PR[GP1:91,1] = PR[GP1:90,1] + 74.643;
   1:  PR[GP1:91,2] = PR[GP1:90,2] + 0.017;
   1:L PR[91] 10mm/sec CNT100;
   1:  PR[GP1:91,1] = PR[GP1:90,1] + 74.277;
   1:  PR[GP1:91,2] = PR[GP1:90,2] + 3.928;
   1:L PR[91] 10mm/sec CNT100;
   1:  PR[GP1:91,1] = PR[GP1:90,1] + 73.537;
   1:  PR[GP1:91,2] = PR[GP1:90,2] + 8.323;
   1:L PR[91] 10mm/sec CNT100;
   1:  PR[GP1:91,1] = PR[GP1:90,1] + 72.473;
   1:  PR[GP1:91,2] = PR[GP1:90,2] + 12.018;
   1:L PR[91] 10mm/sec CNT100;
   1:  PR[GP1:91,1] = PR[GP1:90,1] + 70.730;
   1:  PR[GP1:91,2] = PR[GP1:90,2] + 15.472;
   1:L PR[91] 10mm/sec CNT100;
   1:  PR[GP1:91,1] = PR[GP1:90,1] + 68.527;
   1:  PR[GP1:91,2] = PR[GP1:90,2] + 19.508;
   1:L PR[91] 10mm/sec CNT100;
   1:  PR[GP1:91,1] = PR[GP1:90,1] + 66.247;
   1:  PR[GP1:91,2] = PR[GP1:90,2] + 22.481;
   1:L PR[91] 10mm/sec CNT100;
   1:  PR[GP1:91,1] = PR[GP1:90,1] + 63.417;
   1:  PR[GP1:91,2] = PR[GP1:90,2] + 25.011;
   1:L PR[91] 10mm/sec CNT100;
   1:  PR[GP1:91,1] = PR[GP1:90,1] + 59.902;
   1:  PR[GP1:91,2] = PR[GP1:90,2] + 28.217;
   1:L PR[91] 10mm/sec CNT100;
   1:  PR[GP1:91,1] = PR[GP1:90,1] + 56.829;
   1:  PR[GP1:91,2] = PR[GP1:90,2] + 30.070;
   1:L PR[91] 10mm/sec CNT100;
   1:  PR[GP1:91,1] = PR[GP1:90,1] + 53.394;
   1:  PR[GP1:91,2] = PR[GP1:90,2] + 31.346;
   1:L PR[91] 10mm/sec CNT100;
   1:  PR[GP1:91,1] = PR[GP1:90,1] + 48.813;
   1:  PR[GP1:91,2] = PR[GP1:90,2] + 33.330;
   1:L PR[91] 10mm/sec CNT100;
   1:  PR[GP1:91,1] = PR[GP1:90,1] + 45.461;
   1:  PR[GP1:91,2] = PR[GP1:90,2] + 33.901;
   1:L PR[91] 10mm/sec CNT100;
   1:  PR[GP1:91,1] = PR[GP1:90,1] + 39.912;
   1:  PR[GP1:91,2] = PR[GP1:90,2] + 34.319;
   1:L PR[91] 10mm/sec CNT100;
   1:  PR[GP1:91,1] = PR[GP1:90,1] + 36.754;
   1:  PR[GP1:91,2] = PR[GP1:90,2] + 34.261;
   1:L PR[91] 10mm/sec CNT100;
   1:  PR[GP1:91,1] = PR[GP1:90,1] + 33.649;
   1:  PR[GP1:91,2] = PR[GP1:90,2] + 33.615;
   1:L PR[91] 10mm/sec CNT100;
   1:  PR[GP1:91,1] = PR[GP1:90,1] + 27.852;
   1:  PR[GP1:91,2] = PR[GP1:90,2] + 32.099;
   1:L PR[91] 10mm/sec CNT100;
   1:  PR[GP1:91,1] = PR[GP1:90,1] + 25.219;
   1:  PR[GP1:91,2] = PR[GP1:90,2] + 31.010;
   1:L PR[91] 10mm/sec CNT100;
   1:  PR[GP1:91,1] = PR[GP1:90,1] + 22.802;
   1:  PR[GP1:91,2] = PR[GP1:90,2] + 29.430;
   1:L PR[91] 10mm/sec CNT100;
   1:  PR[GP1:91,1] = PR[GP1:90,1] + 17.427;
   1:  PR[GP1:91,2] = PR[GP1:90,2] + 25.862;
   1:L PR[91] 10mm/sec CNT100;
   1:  PR[GP1:91,1] = PR[GP1:90,1] + 15.600;
   1:  PR[GP1:91,2] = PR[GP1:90,2] + 24.105;
   1:L PR[91] 10mm/sec CNT100;
   1:  PR[GP1:91,1] = PR[GP1:90,1] + 14.095;
   1:  PR[GP1:91,2] = PR[GP1:90,2] + 21.988;
   1:L PR[91] 10mm/sec CNT100;
   1:  PR[GP1:91,1] = PR[GP1:90,1] + 9.893;
   1:  PR[GP1:91,2] = PR[GP1:90,2] + 16.499;
   1:L PR[91] 10mm/sec CNT100;
   1:  PR[GP1:91,1] = PR[GP1:90,1] + 8.936;
   1:  PR[GP1:91,2] = PR[GP1:90,2] + 14.418;
   1:L PR[91] 10mm/sec CNT100;
   1:  PR[GP1:91,1] = PR[GP1:90,1] + 6.578;
   1:  PR[GP1:91,2] = PR[GP1:90,2] + 7.303;
   1:L PR[91] 10mm/sec CNT100;
   1:  PR[GP1:91,1] = PR[GP1:90,1] + 6.161;
   1:  PR[GP1:91,2] = PR[GP1:90,2] + 5.628;
   1:L PR[91] 10mm/sec CNT100;
   1:  PR[GP1:91,1] = PR[GP1:90,1] + 6.191;
   1:  PR[GP1:91,2] = PR[GP1:90,2] + 5.610;
   1:L PR[91] 10mm/sec CNT100;
   1:  PR[GP1:91,1] = PR[GP1:90,1] + 6.135;
   1:  PR[GP1:91,2] = PR[GP1:90,2] + 5.096;
   1:L PR[91] 10mm/sec CNT100;
   1:  PR[GP1:91,1] = PR[GP1:90,1] + 5.787;
   1:  PR[GP1:91,2] = PR[GP1:90,2] + 4.267;
   1:L PR[91] 10mm/sec CNT100;
   1:  PR[GP1:91,1] = PR[GP1:90,1] + 5.347;
   1:  PR[GP1:91,2] = PR[GP1:90,2] + 3.420;
   1:L PR[91] 10mm/sec CNT100;
   1:  PR[GP1:91,1] = PR[GP1:90,1] + 4.785;
   1:  PR[GP1:91,2] = PR[GP1:90,2] + 2.405;
   1:L PR[91] 10mm/sec CNT100;
   1:  PR[GP1:91,1] = PR[GP1:90,1] + 4.215;
   1:  PR[GP1:91,2] = PR[GP1:90,2] + 1.786;
   1:L PR[91] 10mm/sec CNT100;
   1:  PR[GP1:91,1] = PR[GP1:90,1] + 3.354;
   1:  PR[GP1:91,2] = PR[GP1:90,2] + 1.192;
   1:L PR[91] 10mm/sec CNT100;
   1:  PR[GP1:91,1] = PR[GP1:90,1] + 2.358;
   1:  PR[GP1:91,2] = PR[GP1:90,2] + 0.823;
   1:L PR[91] 10mm/sec CNT100;
   1:  PR[GP1:91,1] = PR[GP1:90,1] + 1.738;
   1:  PR[GP1:91,2] = PR[GP1:90,2] + 0.658;
   1:L PR[91] 10mm/sec CNT100;
   1:  PR[GP1:91,1] = PR[GP1:90,1] + 0.647;
   1:  PR[GP1:91,2] = PR[GP1:90,2] + 0.396;
   1:L PR[91] 10mm/sec CNT100;
   1:  PR[GP1:91,1] = PR[GP1:90,1] + 0.130;
   1:L PR[91] 10mm/sec CNT100;
   1:  PR[GP1:91,1] = PR[GP1:90,1] + -0.033;
   1:  PR[GP1:91,2] = PR[GP1:90,2] + 0.440;
   1:  PR[GP1:91,3] = PR[GP1:90,3] + 14.630;
   1:L PR[91] 10mm/sec CNT100;
   1:  PR[GP1:91,1] = PR[GP1:90,1] + -3.284;
   1:  PR[GP1:91,2] = PR[GP1:90,2] + 1.727;
   1:L PR[91] 10mm/sec CNT100;
   1:  PR[GP1:91,1] = PR[GP1:90,1] + -3.497;
   1:  PR[GP1:91,2] = PR[GP1:90,2] + 2.112;
   1:L PR[91] 10mm/sec CNT100;
   1:  PR[GP1:91,1] = PR[GP1:90,1] + -3.564;
   1:  PR[GP1:91,2] = PR[GP1:90,2] + 2.173;
   1:L PR[91] 10mm/sec CNT100;
   1:  PR[GP1:91,1] = PR[GP1:90,1] + -3.820;
   1:  PR[GP1:91,2] = PR[GP1:90,2] + 2.589;
   1:L PR[91] 10mm/sec CNT100;
   1:  PR[GP1:91,1] = PR[GP1:90,1] + -5.162;
   1:  PR[GP1:91,2] = PR[GP1:90,2] + 5.067;
   1:L PR[91] 10mm/sec CNT100;
   1:  PR[GP1:91,1] = PR[GP1:90,1] + -5.211;
   1:  PR[GP1:91,2] = PR[GP1:90,2] + 5.520;
   1:L PR[91] 10mm/sec CNT100;
   1:  PR[GP1:91,1] = PR[GP1:90,1] + -5.361;
   1:  PR[GP1:91,2] = PR[GP1:90,2] + 6.122;
   1:L PR[91] 10mm/sec CNT100;
   1:  PR[GP1:91,1] = PR[GP1:90,1] + -8.402;
   1:  PR[GP1:91,2] = PR[GP1:90,2] + 15.298;
   1:L PR[91] 10mm/sec CNT100;
   1:  PR[GP1:91,1] = PR[GP1:90,1] + -8.866;
   1:  PR[GP1:91,2] = PR[GP1:90,2] + 16.308;
   1:L PR[91] 10mm/sec CNT100;
   1:  PR[GP1:91,1] = PR[GP1:90,1] + -9.523;
   1:  PR[GP1:91,2] = PR[GP1:90,2] + 17.232;
   1:L PR[91] 10mm/sec CNT100;
   1:  PR[GP1:91,1] = PR[GP1:90,1] + -15.131;
   1:  PR[GP1:91,2] = PR[GP1:90,2] + 24.573;
   1:L PR[91] 10mm/sec CNT100;
   1:  PR[GP1:91,1] = PR[GP1:90,1] + -16.160;
   1:  PR[GP1:91,2] = PR[GP1:90,2] + 25.563;
   1:L PR[91] 10mm/sec CNT100;
   1:  PR[GP1:91,1] = PR[GP1:90,1] + -24.649;
   1:  PR[GP1:91,2] = PR[GP1:90,2] + 31.182;
   1:L PR[91] 10mm/sec CNT100;
   1:  PR[GP1:91,1] = PR[GP1:90,1] + -26.315;
   1:  PR[GP1:91,2] = PR[GP1:90,2] + 31.871;
   1:L PR[91] 10mm/sec CNT100;
   1:  PR[GP1:91,1] = PR[GP1:90,1] + -28.151;
   1:  PR[GP1:91,2] = PR[GP1:90,2] + 32.253;
   1:L PR[91] 10mm/sec CNT100;
   1:  PR[GP1:91,1] = PR[GP1:90,1] + -36.000;
   1:  PR[GP1:91,2] = PR[GP1:90,2] + 34.285;
   1:L PR[91] 10mm/sec CNT100;
   1:  PR[GP1:91,1] = PR[GP1:90,1] + -38.199;
   1:  PR[GP1:91,2] = PR[GP1:90,2] + 34.325;
   1:L PR[91] 10mm/sec CNT100;
   1:  PR[GP1:91,1] = PR[GP1:90,1] + -45.356;
   1:  PR[GP1:91,2] = PR[GP1:90,2] + 33.787;
   1:L PR[91] 10mm/sec CNT100;
   1:  PR[GP1:91,1] = PR[GP1:90,1] + -47.866;
   1:  PR[GP1:91,2] = PR[GP1:90,2] + 33.359;
   1:L PR[91] 10mm/sec CNT100;
   1:  PR[GP1:91,1] = PR[GP1:90,1] + -50.265;
   1:  PR[GP1:91,2] = PR[GP1:90,2] + 32.468;
   1:L PR[91] 10mm/sec CNT100;
   1:  PR[GP1:91,1] = PR[GP1:90,1] + -56.421;
   1:  PR[GP1:91,2] = PR[GP1:90,2] + 29.816;
   1:L PR[91] 10mm/sec CNT100;
   1:  PR[GP1:91,1] = PR[GP1:90,1] + -58.815;
   1:  PR[GP1:91,2] = PR[GP1:90,2] + 28.372;
   1:L PR[91] 10mm/sec CNT100;
   1:  PR[GP1:91,1] = PR[GP1:90,1] + -60.928;
   1:  PR[GP1:91,2] = PR[GP1:90,2] + 26.483;
   1:L PR[91] 10mm/sec CNT100;
   1:  PR[GP1:91,1] = PR[GP1:90,1] + -65.601;
   1:  PR[GP1:91,2] = PR[GP1:90,2] + 22.225;
   1:L PR[91] 10mm/sec CNT100;
   1:  PR[GP1:91,1] = PR[GP1:90,1] + -67.408;
   1:  PR[GP1:91,2] = PR[GP1:90,2] + 19.868;
   1:L PR[91] 10mm/sec CNT100;
   1:  PR[GP1:91,1] = PR[GP1:90,1] + -68.775;
   1:  PR[GP1:91,2] = PR[GP1:90,2] + 17.161;
   1:L PR[91] 10mm/sec CNT100;
   1:  PR[GP1:91,1] = PR[GP1:90,1] + -71.667;
   1:  PR[GP1:91,2] = PR[GP1:90,2] + 11.851;
   1:L PR[91] 10mm/sec CNT100;
   1:  PR[GP1:91,1] = PR[GP1:90,1] + -72.516;
   1:  PR[GP1:91,2] = PR[GP1:90,2] + 8.904;
   1:L PR[91] 10mm/sec CNT100;
   1:  PR[GP1:91,1] = PR[GP1:90,1] + -72.811;
   1:  PR[GP1:91,2] = PR[GP1:90,2] + 5.762;
   1:L PR[91] 10mm/sec CNT100;
   1:  PR[GP1:91,1] = PR[GP1:90,1] + -73.776;
   1:  PR[GP1:91,2] = PR[GP1:90,2] + -0.026;
   1:L PR[91] 10mm/sec CNT100;
   1:  PR[GP1:91,1] = PR[GP1:90,1] + -73.477;
   1:  PR[GP1:91,2] = PR[GP1:90,2] + -3.221;
   1:L PR[91] 10mm/sec CNT100;
   1:  PR[GP1:91,1] = PR[GP1:90,1] + -72.522;
   1:  PR[GP1:91,2] = PR[GP1:90,2] + -8.891;
   1:L PR[91] 10mm/sec CNT100;
   1:  PR[GP1:91,1] = PR[GP1:90,1] + -71.664;
   1:  PR[GP1:91,2] = PR[GP1:90,2] + -11.869;
   1:L PR[91] 10mm/sec CNT100;
   1:  PR[GP1:91,1] = PR[GP1:90,1] + -70.257;
   1:  PR[GP1:91,2] = PR[GP1:90,2] + -14.658;
   1:L PR[91] 10mm/sec CNT100;
   1:  PR[GP1:91,1] = PR[GP1:90,1] + -67.414;
   1:  PR[GP1:91,2] = PR[GP1:90,2] + -19.869;
   1:L PR[91] 10mm/sec CNT100;
   1:  PR[GP1:91,1] = PR[GP1:90,1] + -65.603;
   1:  PR[GP1:91,2] = PR[GP1:90,2] + -22.231;
   1:L PR[91] 10mm/sec CNT100;
   1:  PR[GP1:91,1] = PR[GP1:90,1] + -63.347;
   1:  PR[GP1:91,2] = PR[GP1:90,2] + -24.248;
   1:L PR[91] 10mm/sec CNT100;
   1:  PR[GP1:91,1] = PR[GP1:90,1] + -58.813;
   1:  PR[GP1:91,2] = PR[GP1:90,2] + -28.382;
   1:L PR[91] 10mm/sec CNT100;
   1:  PR[GP1:91,1] = PR[GP1:90,1] + -56.434;
   1:  PR[GP1:91,2] = PR[GP1:90,2] + -29.817;
   1:L PR[91] 10mm/sec CNT100;
   1:  PR[GP1:91,1] = PR[GP1:90,1] + -53.760;
   1:  PR[GP1:91,2] = PR[GP1:90,2] + -30.810;
   1:L PR[91] 10mm/sec CNT100;
   1:  PR[GP1:91,1] = PR[GP1:90,1] + -47.850;
   1:  PR[GP1:91,2] = PR[GP1:90,2] + -33.371;
   1:L PR[91] 10mm/sec CNT100;
   1:  PR[GP1:91,1] = PR[GP1:90,1] + -45.356;
   1:  PR[GP1:91,2] = PR[GP1:90,2] + -33.796;
   1:L PR[91] 10mm/sec CNT100;
   1:  PR[GP1:91,1] = PR[GP1:90,1] + -38.199;
   1:  PR[GP1:91,2] = PR[GP1:90,2] + -34.334;
   1:L PR[91] 10mm/sec CNT100;
   1:  PR[GP1:91,1] = PR[GP1:90,1] + -35.985;
   1:  PR[GP1:91,2] = PR[GP1:90,2] + -34.294;
   1:L PR[91] 10mm/sec CNT100;
   1:  PR[GP1:91,1] = PR[GP1:90,1] + -33.805;
   1:  PR[GP1:91,2] = PR[GP1:90,2] + -33.840;
   1:L PR[91] 10mm/sec CNT100;
   1:  PR[GP1:91,1] = PR[GP1:90,1] + -26.329;
   1:  PR[GP1:91,2] = PR[GP1:90,2] + -31.886;
   1:L PR[91] 10mm/sec CNT100;
   1:  PR[GP1:91,1] = PR[GP1:90,1] + -24.648;
   1:  PR[GP1:91,2] = PR[GP1:90,2] + -31.190;
   1:L PR[91] 10mm/sec CNT100;
   1:  PR[GP1:91,1] = PR[GP1:90,1] + -23.092;
   1:  PR[GP1:91,2] = PR[GP1:90,2] + -30.174;
   1:L PR[91] 10mm/sec CNT100;
   1:  PR[GP1:91,1] = PR[GP1:90,1] + -16.160;
   1:  PR[GP1:91,2] = PR[GP1:90,2] + -25.572;
   1:L PR[91] 10mm/sec CNT100;
   1:  PR[GP1:91,1] = PR[GP1:90,1] + -15.139;
   1:  PR[GP1:91,2] = PR[GP1:90,2] + -24.589;
   1:L PR[91] 10mm/sec CNT100;
   1:  PR[GP1:91,1] = PR[GP1:90,1] + -14.280;
   1:  PR[GP1:91,2] = PR[GP1:90,2] + -23.381;
   1:L PR[91] 10mm/sec CNT100;
   1:  PR[GP1:91,1] = PR[GP1:90,1] + -8.862;
   1:  PR[GP1:91,2] = PR[GP1:90,2] + -16.307;
   1:L PR[91] 10mm/sec CNT100;
   1:  PR[GP1:91,1] = PR[GP1:90,1] + -8.402;
   1:  PR[GP1:91,2] = PR[GP1:90,2] + -15.307;
   1:L PR[91] 10mm/sec CNT100;
   1:  PR[GP1:91,1] = PR[GP1:90,1] + -5.361;
   1:  PR[GP1:91,2] = PR[GP1:90,2] + -6.133;
   1:L PR[91] 10mm/sec CNT100;
   1:  PR[GP1:91,1] = PR[GP1:90,1] + -5.213;
   1:  PR[GP1:91,2] = PR[GP1:90,2] + -5.537;
   1:L PR[91] 10mm/sec CNT100;
   1:  PR[GP1:91,1] = PR[GP1:90,1] + -5.166;
   1:  PR[GP1:91,2] = PR[GP1:90,2] + -5.106;
   1:L PR[91] 10mm/sec CNT100;
   1:  PR[GP1:91,1] = PR[GP1:90,1] + -4.410;
   1:  PR[GP1:91,2] = PR[GP1:90,2] + -3.308;
   1:L PR[91] 10mm/sec CNT100;
   1:  PR[GP1:91,1] = PR[GP1:90,1] + -4.016;
   1:  PR[GP1:91,2] = PR[GP1:90,2] + -2.575;
   1:L PR[91] 10mm/sec CNT100;
   1:  PR[GP1:91,1] = PR[GP1:90,1] + -3.308;
   1:  PR[GP1:91,2] = PR[GP1:90,2] + -1.805;
   1:L PR[91] 10mm/sec CNT100;
   1:  PR[GP1:91,1] = PR[GP1:90,1] + -2.223;
   1:  PR[GP1:91,2] = PR[GP1:90,2] + -1.058;
   1:L PR[91] 10mm/sec CNT100;
   1:  PR[GP1:91,1] = PR[GP1:90,1] + -1.754;
   1:  PR[GP1:91,2] = PR[GP1:90,2] + -0.903;
   1:L PR[91] 10mm/sec CNT100;
   1:  PR[GP1:91,1] = PR[GP1:90,1] + 0.403;
   1:  PR[GP1:91,2] = PR[GP1:90,2] + -0.385;
   1:L PR[91] 10mm/sec CNT100;
   1:  PR[GP1:91,1] = PR[GP1:90,1] + 0.596;
   1:  PR[GP1:91,2] = PR[GP1:90,2] + -0.438;
   1:L PR[91] 10mm/sec CNT100;
   1:  PR[GP1:91,1] = PR[GP1:90,1] + 0.854;
   1:  PR[GP1:91,2] = PR[GP1:90,2] + -0.449;
   1:L PR[91] 10mm/sec CNT100;
   1:  PR[GP1:91,1] = PR[GP1:90,1] + 4.104;
   1:  PR[GP1:91,2] = PR[GP1:90,2] + -1.736;
   1:L PR[91] 10mm/sec CNT100;
   1:  PR[GP1:91,1] = PR[GP1:90,1] + 4.317;
   1:  PR[GP1:91,2] = PR[GP1:90,2] + -2.121;
   1:L PR[91] 10mm/sec CNT100;
   1:  PR[GP1:91,1] = PR[GP1:90,1] + 4.385;
   1:  PR[GP1:91,2] = PR[GP1:90,2] + -2.182;
   1:L PR[91] 10mm/sec CNT100;
   1:  PR[GP1:91,1] = PR[GP1:90,1] + 4.641;
   1:  PR[GP1:91,2] = PR[GP1:90,2] + -2.599;
   1:L PR[91] 10mm/sec CNT100;
   1:  PR[GP1:91,1] = PR[GP1:90,1] + 5.982;
   1:  PR[GP1:91,2] = PR[GP1:90,2] + -5.077;
   1:L PR[91] 10mm/sec CNT100;
   1:  PR[GP1:91,1] = PR[GP1:90,1] + 6.032;
   1:  PR[GP1:91,2] = PR[GP1:90,2] + -5.531;
   1:L PR[91] 10mm/sec CNT100;
   1:  PR[GP1:91,1] = PR[GP1:90,1] + 6.182;
   1:  PR[GP1:91,2] = PR[GP1:90,2] + -6.133;
   1:L PR[91] 10mm/sec CNT100;
   1:  PR[GP1:91,1] = PR[GP1:90,1] + 9.221;
   1:  PR[GP1:91,2] = PR[GP1:90,2] + -15.303;
   1:L PR[91] 10mm/sec CNT100;
   1:  PR[GP1:91,1] = PR[GP1:90,1] + 9.686;
   1:  PR[GP1:91,2] = PR[GP1:90,2] + -16.313;
   1:L PR[91] 10mm/sec CNT100;
   1:  PR[GP1:91,1] = PR[GP1:90,1] + 10.343;
   1:  PR[GP1:91,2] = PR[GP1:90,2] + -17.237;
   1:L PR[91] 10mm/sec CNT100;
   1:  PR[GP1:91,1] = PR[GP1:90,1] + 15.950;
   1:  PR[GP1:91,2] = PR[GP1:90,2] + -24.581;
   1:L PR[91] 10mm/sec CNT100;
   1:  PR[GP1:91,1] = PR[GP1:90,1] + 16.979;
   1:  PR[GP1:91,2] = PR[GP1:90,2] + -25.571;
   1:L PR[91] 10mm/sec CNT100;
   1:  PR[GP1:91,1] = PR[GP1:90,1] + 25.468;
   1:  PR[GP1:91,2] = PR[GP1:90,2] + -31.190;
   1:L PR[91] 10mm/sec CNT100;
   1:  PR[GP1:91,1] = PR[GP1:90,1] + 27.134;
   1:  PR[GP1:91,2] = PR[GP1:90,2] + -31.879;
   1:L PR[91] 10mm/sec CNT100;
   1:  PR[GP1:91,1] = PR[GP1:90,1] + 28.969;
   1:  PR[GP1:91,2] = PR[GP1:90,2] + -32.261;
   1:L PR[91] 10mm/sec CNT100;
   1:  PR[GP1:91,1] = PR[GP1:90,1] + 36.819;
   1:  PR[GP1:91,2] = PR[GP1:90,2] + -34.294;
   1:L PR[91] 10mm/sec CNT100;
   1:  PR[GP1:91,1] = PR[GP1:90,1] + 39.018;
   1:  PR[GP1:91,2] = PR[GP1:90,2] + -34.334;
   1:L PR[91] 10mm/sec CNT100;
   1:  PR[GP1:91,1] = PR[GP1:90,1] + 46.175;
   1:  PR[GP1:91,2] = PR[GP1:90,2] + -33.796;
   1:L PR[91] 10mm/sec CNT100;
   1:  PR[GP1:91,1] = PR[GP1:90,1] + 48.686;
   1:  PR[GP1:91,2] = PR[GP1:90,2] + -33.368;
   1:L PR[91] 10mm/sec CNT100;
   1:  PR[GP1:91,1] = PR[GP1:90,1] + 51.085;
   1:  PR[GP1:91,2] = PR[GP1:90,2] + -32.477;
   1:L PR[91] 10mm/sec CNT100;
   1:  PR[GP1:91,1] = PR[GP1:90,1] + 57.241;
   1:  PR[GP1:91,2] = PR[GP1:90,2] + -29.826;
   1:L PR[91] 10mm/sec CNT100;
   1:  PR[GP1:91,1] = PR[GP1:90,1] + 59.635;
   1:  PR[GP1:91,2] = PR[GP1:90,2] + -28.382;
   1:L PR[91] 10mm/sec CNT100;
   1:  PR[GP1:91,1] = PR[GP1:90,1] + 61.748;
   1:  PR[GP1:91,2] = PR[GP1:90,2] + -26.493;
   1:L PR[91] 10mm/sec CNT100;
   1:  PR[GP1:91,1] = PR[GP1:90,1] + 66.421;
   1:  PR[GP1:91,2] = PR[GP1:90,2] + -22.233;
   1:L PR[91] 10mm/sec CNT100;
   1:  PR[GP1:91,1] = PR[GP1:90,1] + 68.229;
   1:  PR[GP1:91,2] = PR[GP1:90,2] + -19.876;
   1:L PR[91] 10mm/sec CNT100;
   1:  PR[GP1:91,1] = PR[GP1:90,1] + 69.595;
   1:  PR[GP1:91,2] = PR[GP1:90,2] + -17.169;
   1:L PR[91] 10mm/sec CNT100;
   1:  PR[GP1:91,1] = PR[GP1:90,1] + 72.488;
   1:  PR[GP1:91,2] = PR[GP1:90,2] + -11.863;
   1:L PR[91] 10mm/sec CNT100;
   1:  PR[GP1:91,1] = PR[GP1:90,1] + 73.337;
   1:  PR[GP1:91,2] = PR[GP1:90,2] + -8.915;
   1:L PR[91] 10mm/sec CNT100;
   1:  PR[GP1:91,1] = PR[GP1:90,1] + 73.631;
   1:  PR[GP1:91,2] = PR[GP1:90,2] + -5.774;
   1:L PR[91] 10mm/sec CNT100;
   1:  PR[GP1:91,1] = PR[GP1:90,1] + 74.597;
   1:  PR[GP1:91,2] = PR[GP1:90,2] + 0.017;
   1:L PR[91] 10mm/sec CNT100;
   1:  PR[GP1:91,1] = PR[GP1:90,1] + 74.297;
   1:  PR[GP1:91,2] = PR[GP1:90,2] + 3.213;
   1:L PR[91] 10mm/sec CNT100;
   1:  PR[GP1:91,1] = PR[GP1:90,1] + 73.343;
   1:  PR[GP1:91,2] = PR[GP1:90,2] + 8.885;
   1:L PR[91] 10mm/sec CNT100;
   1:  PR[GP1:91,1] = PR[GP1:90,1] + 72.485;
   1:  PR[GP1:91,2] = PR[GP1:90,2] + 11.863;
   1:L PR[91] 10mm/sec CNT100;
   1:  PR[GP1:91,1] = PR[GP1:90,1] + 71.078;
   1:  PR[GP1:91,2] = PR[GP1:90,2] + 14.652;
   1:L PR[91] 10mm/sec CNT100;
   1:  PR[GP1:91,1] = PR[GP1:90,1] + 68.235;
   1:  PR[GP1:91,2] = PR[GP1:90,2] + 19.860;
   1:L PR[91] 10mm/sec CNT100;
   1:  PR[GP1:91,1] = PR[GP1:90,1] + 66.423;
   1:  PR[GP1:91,2] = PR[GP1:90,2] + 22.221;
   1:L PR[91] 10mm/sec CNT100;
   1:  PR[GP1:91,1] = PR[GP1:90,1] + 64.167;
   1:  PR[GP1:91,2] = PR[GP1:90,2] + 24.238;
   1:L PR[91] 10mm/sec CNT100;
   1:  PR[GP1:91,1] = PR[GP1:90,1] + 59.633;
   1:  PR[GP1:91,2] = PR[GP1:90,2] + 28.375;
   1:L PR[91] 10mm/sec CNT100;
   1:  PR[GP1:91,1] = PR[GP1:90,1] + 57.254;
   1:  PR[GP1:91,2] = PR[GP1:90,2] + 29.809;
   1:L PR[91] 10mm/sec CNT100;
   1:  PR[GP1:91,1] = PR[GP1:90,1] + 54.580;
   1:  PR[GP1:91,2] = PR[GP1:90,2] + 30.802;
   1:L PR[91] 10mm/sec CNT100;
   1:  PR[GP1:91,1] = PR[GP1:90,1] + 48.670;
   1:  PR[GP1:91,2] = PR[GP1:90,2] + 33.362;
   1:L PR[91] 10mm/sec CNT100;
   1:  PR[GP1:91,1] = PR[GP1:90,1] + 46.175;
   1:  PR[GP1:91,2] = PR[GP1:90,2] + 33.787;
   1:L PR[91] 10mm/sec CNT100;
   1:  PR[GP1:91,1] = PR[GP1:90,1] + 39.018;
   1:  PR[GP1:91,2] = PR[GP1:90,2] + 34.325;
   1:L PR[91] 10mm/sec CNT100;
   1:  PR[GP1:91,1] = PR[GP1:90,1] + 36.804;
   1:  PR[GP1:91,2] = PR[GP1:90,2] + 34.285;
   1:L PR[91] 10mm/sec CNT100;
   1:  PR[GP1:91,1] = PR[GP1:90,1] + 34.624;
   1:  PR[GP1:91,2] = PR[GP1:90,2] + 33.831;
   1:L PR[91] 10mm/sec CNT100;
   1:  PR[GP1:91,1] = PR[GP1:90,1] + 27.148;
   1:  PR[GP1:91,2] = PR[GP1:90,2] + 31.876;
   1:L PR[91] 10mm/sec CNT100;
   1:  PR[GP1:91,1] = PR[GP1:90,1] + 25.467;
   1:  PR[GP1:91,2] = PR[GP1:90,2] + 31.181;
   1:L PR[91] 10mm/sec CNT100;
   1:  PR[GP1:91,1] = PR[GP1:90,1] + 23.911;
   1:  PR[GP1:91,2] = PR[GP1:90,2] + 30.164;
   1:L PR[91] 10mm/sec CNT100;
   1:  PR[GP1:91,1] = PR[GP1:90,1] + 16.979;
   1:  PR[GP1:91,2] = PR[GP1:90,2] + 25.562;
   1:L PR[91] 10mm/sec CNT100;
   1:  PR[GP1:91,1] = PR[GP1:90,1] + 15.958;
   1:  PR[GP1:91,2] = PR[GP1:90,2] + 24.580;
   1:L PR[91] 10mm/sec CNT100;
   1:  PR[GP1:91,1] = PR[GP1:90,1] + 15.099;
   1:  PR[GP1:91,2] = PR[GP1:90,2] + 23.371;
   1:L PR[91] 10mm/sec CNT100;
   1:  PR[GP1:91,1] = PR[GP1:90,1] + 9.681;
   1:  PR[GP1:91,2] = PR[GP1:90,2] + 16.294;
   1:L PR[91] 10mm/sec CNT100;
   1:  PR[GP1:91,1] = PR[GP1:90,1] + 9.221;
   1:  PR[GP1:91,2] = PR[GP1:90,2] + 15.295;
   1:L PR[91] 10mm/sec CNT100;
   1:  PR[GP1:91,1] = PR[GP1:90,1] + 6.181;
   1:  PR[GP1:91,2] = PR[GP1:90,2] + 6.122;
   1:L PR[91] 10mm/sec CNT100;
   1:  PR[GP1:91,1] = PR[GP1:90,1] + 6.033;
   1:  PR[GP1:91,2] = PR[GP1:90,2] + 5.528;
   1:L PR[91] 10mm/sec CNT100;
   1:  PR[GP1:91,1] = PR[GP1:90,1] + 5.986;
   1:  PR[GP1:91,2] = PR[GP1:90,2] + 5.098;
   1:L PR[91] 10mm/sec CNT100;
   1:  PR[GP1:91,1] = PR[GP1:90,1] + 5.232;
   1:  PR[GP1:91,2] = PR[GP1:90,2] + 3.301;
   1:L PR[91] 10mm/sec CNT100;
   1:  PR[GP1:91,1] = PR[GP1:90,1] + 4.837;
   1:  PR[GP1:91,2] = PR[GP1:90,2] + 2.567;
   1:L PR[91] 10mm/sec CNT100;
   1:  PR[GP1:91,1] = PR[GP1:90,1] + 4.128;
   1:  PR[GP1:91,2] = PR[GP1:90,2] + 1.797;
   1:L PR[91] 10mm/sec CNT100;
   1:  PR[GP1:91,1] = PR[GP1:90,1] + 3.044;
   1:  PR[GP1:91,2] = PR[GP1:90,2] + 1.049;
   1:L PR[91] 10mm/sec CNT100;
   1:  PR[GP1:91,1] = PR[GP1:90,1] + 2.573;
   1:  PR[GP1:91,2] = PR[GP1:90,2] + 0.894;
   1:L PR[91] 10mm/sec CNT100;
   1:  PR[GP1:91,1] = PR[GP1:90,1] + 0.347;
   1:  PR[GP1:91,2] = PR[GP1:90,2] + 0.368;
   1:L PR[91] 10mm/sec CNT100;
   1:  PR[GP1:91,1] = PR[GP1:90,1] + 0.191;
   1:  PR[GP1:91,2] = PR[GP1:90,2] + 0.430;
   1:L PR[91] 10mm/sec CNT100;
   1:  PR[GP1:91,1] = PR[GP1:90,1] + -2.902;
   1:  PR[GP1:91,2] = PR[GP1:90,2] + 1.855;
   1:  PR[GP1:91,3] = PR[GP1:90,3] + 15.960;
   1:L PR[91] 10mm/sec CNT100;
   1:  PR[GP1:91,1] = PR[GP1:90,1] + -3.131;
   1:  PR[GP1:91,2] = PR[GP1:90,2] + 2.042;
   1:L PR[91] 10mm/sec CNT100;
   1:  PR[GP1:91,1] = PR[GP1:90,1] + -5.016;
   1:  PR[GP1:91,2] = PR[GP1:90,2] + 5.352;
   1:L PR[91] 10mm/sec CNT100;
   1:  PR[GP1:91,1] = PR[GP1:90,1] + -8.669;
   1:  PR[GP1:91,2] = PR[GP1:90,2] + 16.121;
   1:L PR[91] 10mm/sec CNT100;
   1:  PR[GP1:91,1] = PR[GP1:90,1] + -15.489;
   1:  PR[GP1:91,2] = PR[GP1:90,2] + 25.048;
   1:L PR[91] 10mm/sec CNT100;
   1:  PR[GP1:91,1] = PR[GP1:90,1] + -15.713;
   1:  PR[GP1:91,2] = PR[GP1:90,2] + 25.264;
   1:L PR[91] 10mm/sec CNT100;
   1:  PR[GP1:91,1] = PR[GP1:90,1] + -24.897;
   1:  PR[GP1:91,2] = PR[GP1:90,2] + 31.353;
   1:L PR[91] 10mm/sec CNT100;
   1:  PR[GP1:91,1] = PR[GP1:90,1] + -25.611;
   1:  PR[GP1:91,2] = PR[GP1:90,2] + 31.648;
   1:L PR[91] 10mm/sec CNT100;
   1:  PR[GP1:91,1] = PR[GP1:90,1] + -26.439;
   1:  PR[GP1:91,2] = PR[GP1:90,2] + 31.820;
   1:L PR[91] 10mm/sec CNT100;
   1:  PR[GP1:91,1] = PR[GP1:90,1] + -36.051;
   1:  PR[GP1:91,2] = PR[GP1:90,2] + 34.309;
   1:L PR[91] 10mm/sec CNT100;
   1:  PR[GP1:91,1] = PR[GP1:90,1] + -37.306;
   1:  PR[GP1:91,2] = PR[GP1:90,2] + 34.332;
   1:L PR[91] 10mm/sec CNT100;
   1:  PR[GP1:91,1] = PR[GP1:90,1] + -46.070;
   1:  PR[GP1:91,2] = PR[GP1:90,2] + 33.672;
   1:L PR[91] 10mm/sec CNT100;
   1:  PR[GP1:91,1] = PR[GP1:90,1] + -47.723;
   1:  PR[GP1:91,2] = PR[GP1:90,2] + 33.391;
   1:L PR[91] 10mm/sec CNT100;
   1:  PR[GP1:91,1] = PR[GP1:90,1] + -49.306;
   1:  PR[GP1:91,2] = PR[GP1:90,2] + 32.802;
   1:L PR[91] 10mm/sec CNT100;
   1:  PR[GP1:91,1] = PR[GP1:90,1] + -56.846;
   1:  PR[GP1:91,2] = PR[GP1:90,2] + 29.554;
   1:L PR[91] 10mm/sec CNT100;
   1:  PR[GP1:91,1] = PR[GP1:90,1] + -58.546;
   1:  PR[GP1:91,2] = PR[GP1:90,2] + 28.530;
   1:L PR[91] 10mm/sec CNT100;
   1:  PR[GP1:91,1] = PR[GP1:90,1] + -60.053;
   1:  PR[GP1:91,2] = PR[GP1:90,2] + 27.182;
   1:L PR[91] 10mm/sec CNT100;
   1:  PR[GP1:91,1] = PR[GP1:90,1] + -65.778;
   1:  PR[GP1:91,2] = PR[GP1:90,2] + 21.965;
   1:L PR[91] 10mm/sec CNT100;
   1:  PR[GP1:91,1] = PR[GP1:90,1] + -67.116;
   1:  PR[GP1:91,2] = PR[GP1:90,2] + 20.220;
   1:L PR[91] 10mm/sec CNT100;
   1:  PR[GP1:91,1] = PR[GP1:90,1] + -68.136;
   1:  PR[GP1:91,2] = PR[GP1:90,2] + 18.200;
   1:L PR[91] 10mm/sec CNT100;
   1:  PR[GP1:91,1] = PR[GP1:90,1] + -71.679;
   1:  PR[GP1:91,2] = PR[GP1:90,2] + 11.696;
   1:L PR[91] 10mm/sec CNT100;
   1:  PR[GP1:91,1] = PR[GP1:90,1] + -72.322;
   1:  PR[GP1:91,2] = PR[GP1:90,2] + 9.464;
   1:L PR[91] 10mm/sec CNT100;
   1:  PR[GP1:91,1] = PR[GP1:90,1] + -72.547;
   1:  PR[GP1:91,2] = PR[GP1:90,2] + 7.065;
   1:L PR[91] 10mm/sec CNT100;
   1:  PR[GP1:91,1] = PR[GP1:90,1] + -73.730;
   1:  PR[GP1:91,2] = PR[GP1:90,2] + -0.026;
   1:L PR[91] 10mm/sec CNT100;
   1:  PR[GP1:91,1] = PR[GP1:90,1] + -73.497;
   1:  PR[GP1:91,2] = PR[GP1:90,2] + -2.506;
   1:L PR[91] 10mm/sec CNT100;
   1:  PR[GP1:91,1] = PR[GP1:90,1] + -72.328;
   1:  PR[GP1:91,2] = PR[GP1:90,2] + -9.452;
   1:L PR[91] 10mm/sec CNT100;
   1:  PR[GP1:91,1] = PR[GP1:90,1] + -71.676;
   1:  PR[GP1:91,2] = PR[GP1:90,2] + -11.714;
   1:L PR[91] 10mm/sec CNT100;
   1:  PR[GP1:91,1] = PR[GP1:90,1] + -70.605;
   1:  PR[GP1:91,2] = PR[GP1:90,2] + -13.837;
   1:L PR[91] 10mm/sec CNT100;
   1:  PR[GP1:91,1] = PR[GP1:90,1] + -67.122;
   1:  PR[GP1:91,2] = PR[GP1:90,2] + -20.221;
   1:L PR[91] 10mm/sec CNT100;
   1:  PR[GP1:91,1] = PR[GP1:90,1] + -65.780;
   1:  PR[GP1:91,2] = PR[GP1:90,2] + -21.972;
   1:L PR[91] 10mm/sec CNT100;
   1:  PR[GP1:91,1] = PR[GP1:90,1] + -64.098;
   1:  PR[GP1:91,2] = PR[GP1:90,2] + -23.475;
   1:L PR[91] 10mm/sec CNT100;
   1:  PR[GP1:91,1] = PR[GP1:90,1] + -58.543;
   1:  PR[GP1:91,2] = PR[GP1:90,2] + -28.540;
   1:L PR[91] 10mm/sec CNT100;
   1:  PR[GP1:91,1] = PR[GP1:90,1] + -56.860;
   1:  PR[GP1:91,2] = PR[GP1:90,2] + -29.555;
   1:L PR[91] 10mm/sec CNT100;
   1:  PR[GP1:91,1] = PR[GP1:90,1] + -54.946;
   1:  PR[GP1:91,2] = PR[GP1:90,2] + -30.266;
   1:L PR[91] 10mm/sec CNT100;
   1:  PR[GP1:91,1] = PR[GP1:90,1] + -47.707;
   1:  PR[GP1:91,2] = PR[GP1:90,2] + -33.402;
   1:L PR[91] 10mm/sec CNT100;
   1:  PR[GP1:91,1] = PR[GP1:90,1] + -46.070;
   1:  PR[GP1:91,2] = PR[GP1:90,2] + -33.681;
   1:L PR[91] 10mm/sec CNT100;
   1:  PR[GP1:91,1] = PR[GP1:90,1] + -37.306;
   1:  PR[GP1:91,2] = PR[GP1:90,2] + -34.341;
   1:L PR[91] 10mm/sec CNT100;
   1:  PR[GP1:91,1] = PR[GP1:90,1] + -36.036;
   1:  PR[GP1:91,2] = PR[GP1:90,2] + -34.318;
   1:L PR[91] 10mm/sec CNT100;
   1:  PR[GP1:91,1] = PR[GP1:90,1] + -34.780;
   1:  PR[GP1:91,2] = PR[GP1:90,2] + -34.056;
   1:L PR[91] 10mm/sec CNT100;
   1:  PR[GP1:91,1] = PR[GP1:90,1] + -25.625;
   1:  PR[GP1:91,2] = PR[GP1:90,2] + -31.663;
   1:L PR[91] 10mm/sec CNT100;
   1:  PR[GP1:91,1] = PR[GP1:90,1] + -24.897;
   1:  PR[GP1:91,2] = PR[GP1:90,2] + -31.361;
   1:L PR[91] 10mm/sec CNT100;
   1:  PR[GP1:91,1] = PR[GP1:90,1] + -15.713;
   1:  PR[GP1:91,2] = PR[GP1:90,2] + -25.273;
   1:L PR[91] 10mm/sec CNT100;
   1:  PR[GP1:91,1] = PR[GP1:90,1] + -15.496;
   1:  PR[GP1:91,2] = PR[GP1:90,2] + -25.064;
   1:L PR[91] 10mm/sec CNT100;
   1:  PR[GP1:91,1] = PR[GP1:90,1] + -15.284;
   1:  PR[GP1:91,2] = PR[GP1:90,2] + -24.765;
   1:L PR[91] 10mm/sec CNT100;
   1:  PR[GP1:91,1] = PR[GP1:90,1] + -8.669;
   1:  PR[GP1:91,2] = PR[GP1:90,2] + -16.129;
   1:L PR[91] 10mm/sec CNT100;
   1:  PR[GP1:91,1] = PR[GP1:90,1] + -5.033;
   1:  PR[GP1:91,2] = PR[GP1:90,2] + -5.411;
   1:L PR[91] 10mm/sec CNT100;
   1:  PR[GP1:91,1] = PR[GP1:90,1] + -4.722;
   1:  PR[GP1:91,2] = PR[GP1:90,2] + -4.538;
   1:L PR[91] 10mm/sec CNT100;
   1:  PR[GP1:91,1] = PR[GP1:90,1] + -4.045;
   1:  PR[GP1:91,2] = PR[GP1:90,2] + -2.946;
   1:L PR[91] 10mm/sec CNT100;
   1:  PR[GP1:91,1] = PR[GP1:90,1] + -3.559;
   1:  PR[GP1:91,2] = PR[GP1:90,2] + -2.518;
   1:L PR[91] 10mm/sec CNT100;
   1:  PR[GP1:91,1] = PR[GP1:90,1] + -2.954;
   1:  PR[GP1:91,2] = PR[GP1:90,2] + -1.894;
   1:L PR[91] 10mm/sec CNT100;
   1:  PR[GP1:91,1] = PR[GP1:90,1] + -1.938;
   1:  PR[GP1:91,2] = PR[GP1:90,2] + -1.389;
   1:L PR[91] 10mm/sec CNT100;
   1:  PR[GP1:91,1] = PR[GP1:90,1] + -1.147;
   1:  PR[GP1:91,2] = PR[GP1:90,2] + -0.940;
   1:L PR[91] 10mm/sec CNT100;
   1:  PR[GP1:91,1] = PR[GP1:90,1] + 0.073;
   1:  PR[GP1:91,2] = PR[GP1:90,2] + -0.669;
   1:L PR[91] 10mm/sec CNT100;
   1:  PR[GP1:91,1] = PR[GP1:90,1] + 0.335;
   1:  PR[GP1:91,2] = PR[GP1:90,2] + -0.667;
   1:L PR[91] 10mm/sec CNT100;
   1:  PR[GP1:91,1] = PR[GP1:90,1] + 3.723;
   1:  PR[GP1:91,2] = PR[GP1:90,2] + -1.864;
   1:L PR[91] 10mm/sec CNT100;
   1:  PR[GP1:91,1] = PR[GP1:90,1] + 3.952;
   1:  PR[GP1:91,2] = PR[GP1:90,2] + -2.052;
   1:L PR[91] 10mm/sec CNT100;
   1:  PR[GP1:91,1] = PR[GP1:90,1] + 5.324;
   1:  PR[GP1:91,2] = PR[GP1:90,2] + -4.467;
   1:L PR[91] 10mm/sec CNT100;
   1:  PR[GP1:91,1] = PR[GP1:90,1] + 5.682;
   1:  PR[GP1:91,2] = PR[GP1:90,2] + -5.148;
   1:L PR[91] 10mm/sec CNT100;
   1:  PR[GP1:91,1] = PR[GP1:90,1] + 5.818;
   1:  PR[GP1:91,2] = PR[GP1:90,2] + -5.308;
   1:L PR[91] 10mm/sec CNT100;
   1:  PR[GP1:91,1] = PR[GP1:90,1] + 9.489;
   1:  PR[GP1:91,2] = PR[GP1:90,2] + -16.125;
   1:L PR[91] 10mm/sec CNT100;
   1:  PR[GP1:91,1] = PR[GP1:90,1] + 16.307;
   1:  PR[GP1:91,2] = PR[GP1:90,2] + -25.056;
   1:L PR[91] 10mm/sec CNT100;
   1:  PR[GP1:91,1] = PR[GP1:90,1] + 16.532;
   1:  PR[GP1:91,2] = PR[GP1:90,2] + -25.272;
   1:L PR[91] 10mm/sec CNT100;
   1:  PR[GP1:91,1] = PR[GP1:90,1] + 25.716;
   1:  PR[GP1:91,2] = PR[GP1:90,2] + -31.360;
   1:L PR[91] 10mm/sec CNT100;
   1:  PR[GP1:91,1] = PR[GP1:90,1] + 26.430;
   1:  PR[GP1:91,2] = PR[GP1:90,2] + -31.656;
   1:L PR[91] 10mm/sec CNT100;
   1:  PR[GP1:91,1] = PR[GP1:90,1] + 27.258;
   1:  PR[GP1:91,2] = PR[GP1:90,2] + -31.828;
   1:L PR[91] 10mm/sec CNT100;
   1:  PR[GP1:91,1] = PR[GP1:90,1] + 36.870;
   1:  PR[GP1:91,2] = PR[GP1:90,2] + -34.318;
   1:L PR[91] 10mm/sec CNT100;
   1:  PR[GP1:91,1] = PR[GP1:90,1] + 38.125;
   1:  PR[GP1:91,2] = PR[GP1:90,2] + -34.341;
   1:L PR[91] 10mm/sec CNT100;
   1:  PR[GP1:91,1] = PR[GP1:90,1] + 46.890;
   1:  PR[GP1:91,2] = PR[GP1:90,2] + -33.681;
   1:L PR[91] 10mm/sec CNT100;
   1:  PR[GP1:91,1] = PR[GP1:90,1] + 48.543;
   1:  PR[GP1:91,2] = PR[GP1:90,2] + -33.400;
   1:L PR[91] 10mm/sec CNT100;
   1:  PR[GP1:91,1] = PR[GP1:90,1] + 50.126;
   1:  PR[GP1:91,2] = PR[GP1:90,2] + -32.811;
   1:L PR[91] 10mm/sec CNT100;
   1:  PR[GP1:91,1] = PR[GP1:90,1] + 57.666;
   1:  PR[GP1:91,2] = PR[GP1:90,2] + -29.564;
   1:L PR[91] 10mm/sec CNT100;
   1:  PR[GP1:91,1] = PR[GP1:90,1] + 59.366;
   1:  PR[GP1:91,2] = PR[GP1:90,2] + -28.540;
   1:L PR[91] 10mm/sec CNT100;
   1:  PR[GP1:91,1] = PR[GP1:90,1] + 60.873;
   1:  PR[GP1:91,2] = PR[GP1:90,2] + -27.191;
   1:L PR[91] 10mm/sec CNT100;
   1:  PR[GP1:91,1] = PR[GP1:90,1] + 66.598;
   1:  PR[GP1:91,2] = PR[GP1:90,2] + -21.973;
   1:L PR[91] 10mm/sec CNT100;
   1:  PR[GP1:91,1] = PR[GP1:90,1] + 67.937;
   1:  PR[GP1:91,2] = PR[GP1:90,2] + -20.228;
   1:L PR[91] 10mm/sec CNT100;
   1:  PR[GP1:91,1] = PR[GP1:90,1] + 68.956;
   1:  PR[GP1:91,2] = PR[GP1:90,2] + -18.208;
   1:L PR[91] 10mm/sec CNT100;
   1:  PR[GP1:91,1] = PR[GP1:90,1] + 72.500;
   1:  PR[GP1:91,2] = PR[GP1:90,2] + -11.708;
   1:L PR[91] 10mm/sec CNT100;
   1:  PR[GP1:91,1] = PR[GP1:90,1] + 73.142;
   1:  PR[GP1:91,2] = PR[GP1:90,2] + -9.476;
   1:L PR[91] 10mm/sec CNT100;
   1:  PR[GP1:91,1] = PR[GP1:90,1] + 73.367;
   1:  PR[GP1:91,2] = PR[GP1:90,2] + -7.077;
   1:L PR[91] 10mm/sec CNT100;
   1:  PR[GP1:91,1] = PR[GP1:90,1] + 74.550;
   1:  PR[GP1:91,2] = PR[GP1:90,2] + 0.017;
   1:L PR[91] 10mm/sec CNT100;
   1:  PR[GP1:91,1] = PR[GP1:90,1] + 74.318;
   1:  PR[GP1:91,2] = PR[GP1:90,2] + 2.497;
   1:L PR[91] 10mm/sec CNT100;
   1:  PR[GP1:91,1] = PR[GP1:90,1] + 73.148;
   1:  PR[GP1:91,2] = PR[GP1:90,2] + 9.446;
   1:L PR[91] 10mm/sec CNT100;
   1:  PR[GP1:91,1] = PR[GP1:90,1] + 72.497;
   1:  PR[GP1:91,2] = PR[GP1:90,2] + 11.708;
   1:L PR[91] 10mm/sec CNT100;
   1:  PR[GP1:91,1] = PR[GP1:90,1] + 71.426;
   1:  PR[GP1:91,2] = PR[GP1:90,2] + 13.831;
   1:L PR[91] 10mm/sec CNT100;
   1:  PR[GP1:91,1] = PR[GP1:90,1] + 67.943;
   1:  PR[GP1:91,2] = PR[GP1:90,2] + 20.211;
   1:L PR[91] 10mm/sec CNT100;
   1:  PR[GP1:91,1] = PR[GP1:90,1] + 66.600;
   1:  PR[GP1:91,2] = PR[GP1:90,2] + 21.962;
   1:L PR[91] 10mm/sec CNT100;
   1:  PR[GP1:91,1] = PR[GP1:90,1] + 64.918;
   1:  PR[GP1:91,2] = PR[GP1:90,2] + 23.465;
   1:L PR[91] 10mm/sec CNT100;
   1:  PR[GP1:91,1] = PR[GP1:90,1] + 59.363;
   1:  PR[GP1:91,2] = PR[GP1:90,2] + 28.532;
   1:L PR[91] 10mm/sec CNT100;
   1:  PR[GP1:91,1] = PR[GP1:90,1] + 57.680;
   1:  PR[GP1:91,2] = PR[GP1:90,2] + 29.547;
   1:L PR[91] 10mm/sec CNT100;
   1:  PR[GP1:91,1] = PR[GP1:90,1] + 55.766;
   1:  PR[GP1:91,2] = PR[GP1:90,2] + 30.258;
   1:L PR[91] 10mm/sec CNT100;
   1:  PR[GP1:91,1] = PR[GP1:90,1] + 48.527;
   1:  PR[GP1:91,2] = PR[GP1:90,2] + 33.393;
   1:L PR[91] 10mm/sec CNT100;
   1:  PR[GP1:91,1] = PR[GP1:90,1] + 46.890;
   1:  PR[GP1:91,2] = PR[GP1:90,2] + 33.672;
   1:L PR[91] 10mm/sec CNT100;
   1:  PR[GP1:91,1] = PR[GP1:90,1] + 38.125;
   1:  PR[GP1:91,2] = PR[GP1:90,2] + 34.332;
   1:L PR[91] 10mm/sec CNT100;
   1:  PR[GP1:91,1] = PR[GP1:90,1] + 36.855;
   1:  PR[GP1:91,2] = PR[GP1:90,2] + 34.309;
   1:L PR[91] 10mm/sec CNT100;
   1:  PR[GP1:91,1] = PR[GP1:90,1] + 35.599;
   1:  PR[GP1:91,2] = PR[GP1:90,2] + 34.047;
   1:L PR[91] 10mm/sec CNT100;
   1:  PR[GP1:91,1] = PR[GP1:90,1] + 26.444;
   1:  PR[GP1:91,2] = PR[GP1:90,2] + 31.653;
   1:L PR[91] 10mm/sec CNT100;
   1:  PR[GP1:91,1] = PR[GP1:90,1] + 25.716;
   1:  PR[GP1:91,2] = PR[GP1:90,2] + 31.351;
   1:L PR[91] 10mm/sec CNT100;
   1:  PR[GP1:91,1] = PR[GP1:90,1] + 16.532;
   1:  PR[GP1:91,2] = PR[GP1:90,2] + 25.263;
   1:L PR[91] 10mm/sec CNT100;
   1:  PR[GP1:91,1] = PR[GP1:90,1] + 16.315;
   1:  PR[GP1:91,2] = PR[GP1:90,2] + 25.054;
   1:L PR[91] 10mm/sec CNT100;
   1:  PR[GP1:91,1] = PR[GP1:90,1] + 16.103;
   1:  PR[GP1:91,2] = PR[GP1:90,2] + 24.755;
   1:L PR[91] 10mm/sec CNT100;
   1:  PR[GP1:91,1] = PR[GP1:90,1] + 9.488;
   1:  PR[GP1:91,2] = PR[GP1:90,2] + 16.116;
   1:L PR[91] 10mm/sec CNT100;
   1:  PR[GP1:91,1] = PR[GP1:90,1] + 5.853;
   1:  PR[GP1:91,2] = PR[GP1:90,2] + 5.403;
   1:L PR[91] 10mm/sec CNT100;
   1:  PR[GP1:91,1] = PR[GP1:90,1] + 5.542;
   1:  PR[GP1:91,2] = PR[GP1:90,2] + 4.531;
   1:L PR[91] 10mm/sec CNT100;
   1:  PR[GP1:91,1] = PR[GP1:90,1] + 4.866;
   1:  PR[GP1:91,2] = PR[GP1:90,2] + 2.937;
   1:L PR[91] 10mm/sec CNT100;
   1:  PR[GP1:91,1] = PR[GP1:90,1] + 4.380;
   1:  PR[GP1:91,2] = PR[GP1:90,2] + 2.509;
   1:L PR[91] 10mm/sec CNT100;
   1:  PR[GP1:91,1] = PR[GP1:90,1] + 3.774;
   1:  PR[GP1:91,2] = PR[GP1:90,2] + 1.885;
   1:L PR[91] 10mm/sec CNT100;
   1:  PR[GP1:91,1] = PR[GP1:90,1] + 2.759;
   1:  PR[GP1:91,2] = PR[GP1:90,2] + 1.380;
   1:L PR[91] 10mm/sec CNT100;
   1:  PR[GP1:91,1] = PR[GP1:90,1] + 1.967;
   1:  PR[GP1:91,2] = PR[GP1:90,2] + 0.931;
   1:L PR[91] 10mm/sec CNT100;
   1:  PR[GP1:91,1] = PR[GP1:90,1] + 0.748;
   1:  PR[GP1:91,2] = PR[GP1:90,2] + 0.660;
   1:L PR[91] 10mm/sec CNT100;
   1:  PR[GP1:91,1] = PR[GP1:90,1] + 0.486;
   1:  PR[GP1:91,2] = PR[GP1:90,2] + 0.658;
   1:L PR[91] 10mm/sec CNT100;
   1:  PR[GP1:91,1] = PR[GP1:90,1] + -0.489;
   1:  PR[GP1:91,2] = PR[GP1:90,2] + 1.445;
   1:  PR[GP1:91,3] = PR[GP1:90,3] + 17.290;
   1:L PR[91] 10mm/sec CNT100;
   1:  PR[GP1:91,1] = PR[GP1:90,1] + -0.834;
   1:  PR[GP1:91,2] = PR[GP1:90,2] + 1.594;
   1:L PR[91] 10mm/sec CNT100;
   1:  PR[GP1:91,1] = PR[GP1:90,1] + -2.634;
   1:  PR[GP1:91,2] = PR[GP1:90,2] + 2.244;
   1:L PR[91] 10mm/sec CNT100;
   1:  PR[GP1:91,1] = PR[GP1:90,1] + -4.963;
   1:  PR[GP1:91,2] = PR[GP1:90,2] + 6.311;
   1:L PR[91] 10mm/sec CNT100;
   1:  PR[GP1:91,1] = PR[GP1:90,1] + -7.913;
   1:  PR[GP1:91,2] = PR[GP1:90,2] + 15.001;
   1:L PR[91] 10mm/sec CNT100;
   1:  PR[GP1:91,1] = PR[GP1:90,1] + -8.812;
   1:  PR[GP1:91,2] = PR[GP1:90,2] + 16.799;
   1:L PR[91] 10mm/sec CNT100;
   1:  PR[GP1:91,1] = PR[GP1:90,1] + -14.903;
   1:  PR[GP1:91,2] = PR[GP1:90,2] + 24.619;
   1:L PR[91] 10mm/sec CNT100;
   1:  PR[GP1:91,1] = PR[GP1:90,1] + -15.727;
   1:  PR[GP1:91,2] = PR[GP1:90,2] + 25.445;
   1:L PR[91] 10mm/sec CNT100;
   1:  PR[GP1:91,1] = PR[GP1:90,1] + -24.933;
   1:  PR[GP1:91,2] = PR[GP1:90,2] + 31.423;
   1:L PR[91] 10mm/sec CNT100;
   1:  PR[GP1:91,1] = PR[GP1:90,1] + -25.079;
   1:  PR[GP1:91,2] = PR[GP1:90,2] + 31.498;
   1:L PR[91] 10mm/sec CNT100;
   1:  PR[GP1:91,1] = PR[GP1:90,1] + -27.678;
   1:  PR[GP1:91,2] = PR[GP1:90,2] + 32.151;
   1:L PR[91] 10mm/sec CNT100;
   1:  PR[GP1:91,1] = PR[GP1:90,1] + -36.102;
   1:  PR[GP1:91,2] = PR[GP1:90,2] + 34.333;
   1:L PR[91] 10mm/sec CNT100;
   1:  PR[GP1:91,1] = PR[GP1:90,1] + -36.413;
   1:  PR[GP1:91,2] = PR[GP1:90,2] + 34.338;
   1:L PR[91] 10mm/sec CNT100;
   1:  PR[GP1:91,1] = PR[GP1:90,1] + -46.785;
   1:  PR[GP1:91,2] = PR[GP1:90,2] + 33.558;
   1:L PR[91] 10mm/sec CNT100;
   1:  PR[GP1:91,1] = PR[GP1:90,1] + -47.580;
   1:  PR[GP1:91,2] = PR[GP1:90,2] + 33.422;
   1:L PR[91] 10mm/sec CNT100;
   1:  PR[GP1:91,1] = PR[GP1:90,1] + -48.348;
   1:  PR[GP1:91,2] = PR[GP1:90,2] + 33.137;
   1:L PR[91] 10mm/sec CNT100;
   1:  PR[GP1:91,1] = PR[GP1:90,1] + -57.272;
   1:  PR[GP1:91,2] = PR[GP1:90,2] + 29.293;
   1:L PR[91] 10mm/sec CNT100;
   1:  PR[GP1:91,1] = PR[GP1:90,1] + -58.276;
   1:  PR[GP1:91,2] = PR[GP1:90,2] + 28.687;
   1:L PR[91] 10mm/sec CNT100;
   1:  PR[GP1:91,1] = PR[GP1:90,1] + -59.179;
   1:  PR[GP1:91,2] = PR[GP1:90,2] + 27.880;
   1:L PR[91] 10mm/sec CNT100;
   1:  PR[GP1:91,1] = PR[GP1:90,1] + -65.955;
   1:  PR[GP1:91,2] = PR[GP1:90,2] + 21.706;
   1:L PR[91] 10mm/sec CNT100;
   1:  PR[GP1:91,1] = PR[GP1:90,1] + -66.824;
   1:  PR[GP1:91,2] = PR[GP1:90,2] + 20.572;
   1:L PR[91] 10mm/sec CNT100;
   1:  PR[GP1:91,1] = PR[GP1:90,1] + -67.497;
   1:  PR[GP1:91,2] = PR[GP1:90,2] + 19.239;
   1:L PR[91] 10mm/sec CNT100;
   1:  PR[GP1:91,1] = PR[GP1:90,1] + -71.691;
   1:  PR[GP1:91,2] = PR[GP1:90,2] + 11.540;
   1:L PR[91] 10mm/sec CNT100;
   1:  PR[GP1:91,1] = PR[GP1:90,1] + -72.127;
   1:  PR[GP1:91,2] = PR[GP1:90,2] + 10.025;
   1:L PR[91] 10mm/sec CNT100;
   1:  PR[GP1:91,1] = PR[GP1:90,1] + -72.283;
   1:  PR[GP1:91,2] = PR[GP1:90,2] + 8.368;
   1:L PR[91] 10mm/sec CNT100;
   1:  PR[GP1:91,1] = PR[GP1:90,1] + -73.683;
   1:  PR[GP1:91,2] = PR[GP1:90,2] + -0.026;
   1:L PR[91] 10mm/sec CNT100;
   1:  PR[GP1:91,1] = PR[GP1:90,1] + -73.518;
   1:  PR[GP1:91,2] = PR[GP1:90,2] + -1.790;
   1:L PR[91] 10mm/sec CNT100;
   1:  PR[GP1:91,1] = PR[GP1:90,1] + -72.133;
   1:  PR[GP1:91,2] = PR[GP1:90,2] + -10.013;
   1:L PR[91] 10mm/sec CNT100;
   1:  PR[GP1:91,1] = PR[GP1:90,1] + -71.688;
   1:  PR[GP1:91,2] = PR[GP1:90,2] + -11.558;
   1:L PR[91] 10mm/sec CNT100;
   1:  PR[GP1:91,1] = PR[GP1:90,1] + -70.953;
   1:  PR[GP1:91,2] = PR[GP1:90,2] + -13.016;
   1:L PR[91] 10mm/sec CNT100;
   1:  PR[GP1:91,1] = PR[GP1:90,1] + -66.830;
   1:  PR[GP1:91,2] = PR[GP1:90,2] + -20.573;
   1:L PR[91] 10mm/sec CNT100;
   1:  PR[GP1:91,1] = PR[GP1:90,1] + -65.956;
   1:  PR[GP1:91,2] = PR[GP1:90,2] + -21.712;
   1:L PR[91] 10mm/sec CNT100;
   1:  PR[GP1:91,1] = PR[GP1:90,1] + -64.849;
   1:  PR[GP1:91,2] = PR[GP1:90,2] + -22.703;
   1:L PR[91] 10mm/sec CNT100;
   1:  PR[GP1:91,1] = PR[GP1:90,1] + -58.274;
   1:  PR[GP1:91,2] = PR[GP1:90,2] + -28.697;
   1:L PR[91] 10mm/sec CNT100;
   1:  PR[GP1:91,1] = PR[GP1:90,1] + -57.285;
   1:  PR[GP1:91,2] = PR[GP1:90,2] + -29.294;
   1:L PR[91] 10mm/sec CNT100;
   1:  PR[GP1:91,1] = PR[GP1:90,1] + -56.133;
   1:  PR[GP1:91,2] = PR[GP1:90,2] + -29.722;
   1:L PR[91] 10mm/sec CNT100;
   1:  PR[GP1:91,1] = PR[GP1:90,1] + -47.564;
   1:  PR[GP1:91,2] = PR[GP1:90,2] + -33.434;
   1:L PR[91] 10mm/sec CNT100;
   1:  PR[GP1:91,1] = PR[GP1:90,1] + -46.785;
   1:  PR[GP1:91,2] = PR[GP1:90,2] + -33.567;
   1:L PR[91] 10mm/sec CNT100;
   1:  PR[GP1:91,1] = PR[GP1:90,1] + -36.413;
   1:  PR[GP1:91,2] = PR[GP1:90,2] + -34.347;
   1:L PR[91] 10mm/sec CNT100;
   1:  PR[GP1:91,1] = PR[GP1:90,1] + -36.087;
   1:  PR[GP1:91,2] = PR[GP1:90,2] + -34.341;
   1:L PR[91] 10mm/sec CNT100;
   1:  PR[GP1:91,1] = PR[GP1:90,1] + -35.755;
   1:  PR[GP1:91,2] = PR[GP1:90,2] + -34.272;
   1:L PR[91] 10mm/sec CNT100;
   1:  PR[GP1:91,1] = PR[GP1:90,1] + -27.679;
   1:  PR[GP1:91,2] = PR[GP1:90,2] + -32.160;
   1:L PR[91] 10mm/sec CNT100;
   1:  PR[GP1:91,1] = PR[GP1:90,1] + -25.079;
   1:  PR[GP1:91,2] = PR[GP1:90,2] + -31.507;
   1:L PR[91] 10mm/sec CNT100;
   1:  PR[GP1:91,1] = PR[GP1:90,1] + -24.933;
   1:  PR[GP1:91,2] = PR[GP1:90,2] + -31.432;
   1:L PR[91] 10mm/sec CNT100;
   1:  PR[GP1:91,1] = PR[GP1:90,1] + -15.727;
   1:  PR[GP1:91,2] = PR[GP1:90,2] + -25.454;
   1:L PR[91] 10mm/sec CNT100;
   1:  PR[GP1:91,1] = PR[GP1:90,1] + -14.903;
   1:  PR[GP1:91,2] = PR[GP1:90,2] + -24.628;
   1:L PR[91] 10mm/sec CNT100;
   1:  PR[GP1:91,1] = PR[GP1:90,1] + -8.812;
   1:  PR[GP1:91,2] = PR[GP1:90,2] + -16.808;
   1:L PR[91] 10mm/sec CNT100;
   1:  PR[GP1:91,1] = PR[GP1:90,1] + -7.914;
   1:  PR[GP1:91,2] = PR[GP1:90,2] + -15.014;
   1:L PR[91] 10mm/sec CNT100;
   1:  PR[GP1:91,1] = PR[GP1:90,1] + -4.980;
   1:  PR[GP1:91,2] = PR[GP1:90,2] + -6.371;
   1:L PR[91] 10mm/sec CNT100;
   1:  PR[GP1:91,1] = PR[GP1:90,1] + -4.084;
   1:  PR[GP1:91,2] = PR[GP1:90,2] + -3.857;
   1:L PR[91] 10mm/sec CNT100;
   1:  PR[GP1:91,1] = PR[GP1:90,1] + -3.238;
   1:  PR[GP1:91,2] = PR[GP1:90,2] + -2.922;
   1:L PR[91] 10mm/sec CNT100;
   1:  PR[GP1:91,1] = PR[GP1:90,1] + -2.608;
   1:  PR[GP1:91,2] = PR[GP1:90,2] + -2.367;
   1:L PR[91] 10mm/sec CNT100;
   1:  PR[GP1:91,1] = PR[GP1:90,1] + -2.371;
   1:  PR[GP1:91,2] = PR[GP1:90,2] + -2.122;
   1:L PR[91] 10mm/sec CNT100;
   1:  PR[GP1:91,1] = PR[GP1:90,1] + -1.937;
   1:  PR[GP1:91,2] = PR[GP1:90,2] + -1.948;
   1:L PR[91] 10mm/sec CNT100;
   1:  PR[GP1:91,1] = PR[GP1:90,1] + -0.652;
   1:  PR[GP1:91,2] = PR[GP1:90,2] + -1.293;
   1:L PR[91] 10mm/sec CNT100;
   1:  PR[GP1:91,1] = PR[GP1:90,1] + 1.309;
   1:  PR[GP1:91,2] = PR[GP1:90,2] + -1.454;
   1:L PR[91] 10mm/sec CNT100;
   1:  PR[GP1:91,1] = PR[GP1:90,1] + 1.654;
   1:  PR[GP1:91,2] = PR[GP1:90,2] + -1.603;
   1:L PR[91] 10mm/sec CNT100;
   1:  PR[GP1:91,1] = PR[GP1:90,1] + 3.456;
   1:  PR[GP1:91,2] = PR[GP1:90,2] + -2.254;
   1:L PR[91] 10mm/sec CNT100;
   1:  PR[GP1:91,1] = PR[GP1:90,1] + 3.914;
   1:  PR[GP1:91,2] = PR[GP1:90,2] + -3.061;
   1:L PR[91] 10mm/sec CNT100;
   1:  PR[GP1:91,1] = PR[GP1:90,1] + 5.340;
   1:  PR[GP1:91,2] = PR[GP1:90,2] + -5.775;
   1:L PR[91] 10mm/sec CNT100;
   1:  PR[GP1:91,1] = PR[GP1:90,1] + 5.763;
   1:  PR[GP1:91,2] = PR[GP1:90,2] + -6.264;
   1:L PR[91] 10mm/sec CNT100;
   1:  PR[GP1:91,1] = PR[GP1:90,1] + 8.732;
   1:  PR[GP1:91,2] = PR[GP1:90,2] + -15.009;
   1:L PR[91] 10mm/sec CNT100;
   1:  PR[GP1:91,1] = PR[GP1:90,1] + 9.630;
   1:  PR[GP1:91,2] = PR[GP1:90,2] + -16.800;
   1:L PR[91] 10mm/sec CNT100;
   1:  PR[GP1:91,1] = PR[GP1:90,1] + 15.721;
   1:  PR[GP1:91,2] = PR[GP1:90,2] + -24.624;
   1:L PR[91] 10mm/sec CNT100;
   1:  PR[GP1:91,1] = PR[GP1:90,1] + 16.545;
   1:  PR[GP1:91,2] = PR[GP1:90,2] + -25.452;
   1:L PR[91] 10mm/sec CNT100;
   1:  PR[GP1:91,1] = PR[GP1:90,1] + 25.750;
   1:  PR[GP1:91,2] = PR[GP1:90,2] + -31.430;
   1:L PR[91] 10mm/sec CNT100;
   1:  PR[GP1:91,1] = PR[GP1:90,1] + 25.897;
   1:  PR[GP1:91,2] = PR[GP1:90,2] + -31.505;
   1:L PR[91] 10mm/sec CNT100;
   1:  PR[GP1:91,1] = PR[GP1:90,1] + 28.499;
   1:  PR[GP1:91,2] = PR[GP1:90,2] + -32.160;
   1:L PR[91] 10mm/sec CNT100;
   1:  PR[GP1:91,1] = PR[GP1:90,1] + 36.920;
   1:  PR[GP1:91,2] = PR[GP1:90,2] + -34.342;
   1:L PR[91] 10mm/sec CNT100;
   1:  PR[GP1:91,1] = PR[GP1:90,1] + 37.231;
   1:  PR[GP1:91,2] = PR[GP1:90,2] + -34.347;
   1:L PR[91] 10mm/sec CNT100;
   1:  PR[GP1:91,1] = PR[GP1:90,1] + 47.605;
   1:  PR[GP1:91,2] = PR[GP1:90,2] + -33.567;
   1:L PR[91] 10mm/sec CNT100;
   1:  PR[GP1:91,1] = PR[GP1:90,1] + 48.400;
   1:  PR[GP1:91,2] = PR[GP1:90,2] + -33.431;
   1:L PR[91] 10mm/sec CNT100;
   1:  PR[GP1:91,1] = PR[GP1:90,1] + 49.167;
   1:  PR[GP1:91,2] = PR[GP1:90,2] + -33.146;
   1:L PR[91] 10mm/sec CNT100;
   1:  PR[GP1:91,1] = PR[GP1:90,1] + 58.092;
   1:  PR[GP1:91,2] = PR[GP1:90,2] + -29.303;
   1:L PR[91] 10mm/sec CNT100;
   1:  PR[GP1:91,1] = PR[GP1:90,1] + 59.096;
   1:  PR[GP1:91,2] = PR[GP1:90,2] + -28.697;
   1:L PR[91] 10mm/sec CNT100;
   1:  PR[GP1:91,1] = PR[GP1:90,1] + 59.999;
   1:  PR[GP1:91,2] = PR[GP1:90,2] + -27.890;
   1:L PR[91] 10mm/sec CNT100;
   1:  PR[GP1:91,1] = PR[GP1:90,1] + 66.775;
   1:  PR[GP1:91,2] = PR[GP1:90,2] + -21.713;
   1:L PR[91] 10mm/sec CNT100;
   1:  PR[GP1:91,1] = PR[GP1:90,1] + 67.645;
   1:  PR[GP1:91,2] = PR[GP1:90,2] + -20.579;
   1:L PR[91] 10mm/sec CNT100;
   1:  PR[GP1:91,1] = PR[GP1:90,1] + 68.317;
   1:  PR[GP1:91,2] = PR[GP1:90,2] + -19.247;
   1:L PR[91] 10mm/sec CNT100;
   1:  PR[GP1:91,1] = PR[GP1:90,1] + 72.512;
   1:  PR[GP1:91,2] = PR[GP1:90,2] + -11.553;
   1:L PR[91] 10mm/sec CNT100;
   1:  PR[GP1:91,1] = PR[GP1:90,1] + 72.948;
   1:  PR[GP1:91,2] = PR[GP1:90,2] + -10.038;
   1:L PR[91] 10mm/sec CNT100;
   1:  PR[GP1:91,1] = PR[GP1:90,1] + 73.103;
   1:  PR[GP1:91,2] = PR[GP1:90,2] + -8.381;
   1:L PR[91] 10mm/sec CNT100;
   1:  PR[GP1:91,1] = PR[GP1:90,1] + 74.504;
   1:  PR[GP1:91,2] = PR[GP1:90,2] + 0.017;
   1:L PR[91] 10mm/sec CNT100;
   1:  PR[GP1:91,1] = PR[GP1:90,1] + 74.338;
   1:  PR[GP1:91,2] = PR[GP1:90,2] + 1.781;
   1:L PR[91] 10mm/sec CNT100;
   1:  PR[GP1:91,1] = PR[GP1:90,1] + 72.954;
   1:  PR[GP1:91,2] = PR[GP1:90,2] + 10.007;
   1:L PR[91] 10mm/sec CNT100;
   1:  PR[GP1:91,1] = PR[GP1:90,1] + 72.509;
   1:  PR[GP1:91,2] = PR[GP1:90,2] + 11.553;
   1:L PR[91] 10mm/sec CNT100;
   1:  PR[GP1:91,1] = PR[GP1:90,1] + 71.773;
   1:  PR[GP1:91,2] = PR[GP1:90,2] + 13.010;
   1:L PR[91] 10mm/sec CNT100;
   1:  PR[GP1:91,1] = PR[GP1:90,1] + 67.651;
   1:  PR[GP1:91,2] = PR[GP1:90,2] + 20.563;
   1:L PR[91] 10mm/sec CNT100;
   1:  PR[GP1:91,1] = PR[GP1:90,1] + 66.777;
   1:  PR[GP1:91,2] = PR[GP1:90,2] + 21.702;
   1:L PR[91] 10mm/sec CNT100;
   1:  PR[GP1:91,1] = PR[GP1:90,1] + 65.669;
   1:  PR[GP1:91,2] = PR[GP1:90,2] + 22.693;
   1:L PR[91] 10mm/sec CNT100;
   1:  PR[GP1:91,1] = PR[GP1:90,1] + 59.093;
   1:  PR[GP1:91,2] = PR[GP1:90,2] + 28.690;
   1:L PR[91] 10mm/sec CNT100;
   1:  PR[GP1:91,1] = PR[GP1:90,1] + 58.105;
   1:  PR[GP1:91,2] = PR[GP1:90,2] + 29.286;
   1:L PR[91] 10mm/sec CNT100;
   1:  PR[GP1:91,1] = PR[GP1:90,1] + 56.952;
   1:  PR[GP1:91,2] = PR[GP1:90,2] + 29.714;
   1:L PR[91] 10mm/sec CNT100;
   1:  PR[GP1:91,1] = PR[GP1:90,1] + 48.384;
   1:  PR[GP1:91,2] = PR[GP1:90,2] + 33.425;
   1:L PR[91] 10mm/sec CNT100;
   1:  PR[GP1:91,1] = PR[GP1:90,1] + 47.605;
   1:  PR[GP1:91,2] = PR[GP1:90,2] + 33.558;
   1:L PR[91] 10mm/sec CNT100;
   1:  PR[GP1:91,1] = PR[GP1:90,1] + 37.232;
   1:  PR[GP1:91,2] = PR[GP1:90,2] + 34.338;
   1:L PR[91] 10mm/sec CNT100;
   1:  PR[GP1:91,1] = PR[GP1:90,1] + 36.906;
   1:  PR[GP1:91,2] = PR[GP1:90,2] + 34.332;
   1:L PR[91] 10mm/sec CNT100;
   1:  PR[GP1:91,1] = PR[GP1:90,1] + 36.574;
   1:  PR[GP1:91,2] = PR[GP1:90,2] + 34.264;
   1:L PR[91] 10mm/sec CNT100;
   1:  PR[GP1:91,1] = PR[GP1:90,1] + 28.499;
   1:  PR[GP1:91,2] = PR[GP1:90,2] + 32.151;
   1:L PR[91] 10mm/sec CNT100;
   1:  PR[GP1:91,1] = PR[GP1:90,1] + 25.897;
   1:  PR[GP1:91,2] = PR[GP1:90,2] + 31.496;
   1:L PR[91] 10mm/sec CNT100;
   1:  PR[GP1:91,1] = PR[GP1:90,1] + 25.750;
   1:  PR[GP1:91,2] = PR[GP1:90,2] + 31.421;
   1:L PR[91] 10mm/sec CNT100;
   1:  PR[GP1:91,1] = PR[GP1:90,1] + 16.545;
   1:  PR[GP1:91,2] = PR[GP1:90,2] + 25.444;
   1:L PR[91] 10mm/sec CNT100;
   1:  PR[GP1:91,1] = PR[GP1:90,1] + 15.721;
   1:  PR[GP1:91,2] = PR[GP1:90,2] + 24.615;
   1:L PR[91] 10mm/sec CNT100;
   1:  PR[GP1:91,1] = PR[GP1:90,1] + 9.630;
   1:  PR[GP1:91,2] = PR[GP1:90,2] + 16.791;
   1:L PR[91] 10mm/sec CNT100;
   1:  PR[GP1:91,1] = PR[GP1:90,1] + 8.731;
   1:  PR[GP1:91,2] = PR[GP1:90,2] + 14.996;
   1:L PR[91] 10mm/sec CNT100;
   1:  PR[GP1:91,1] = PR[GP1:90,1] + 5.799;
   1:  PR[GP1:91,2] = PR[GP1:90,2] + 6.362;
   1:L PR[91] 10mm/sec CNT100;
   1:  PR[GP1:91,1] = PR[GP1:90,1] + 4.904;
   1:  PR[GP1:91,2] = PR[GP1:90,2] + 3.847;
   1:L PR[91] 10mm/sec CNT100;
   1:  PR[GP1:91,1] = PR[GP1:90,1] + 4.059;
   1:  PR[GP1:91,2] = PR[GP1:90,2] + 2.914;
   1:L PR[91] 10mm/sec CNT100;
   1:  PR[GP1:91,1] = PR[GP1:90,1] + 3.429;
   1:  PR[GP1:91,2] = PR[GP1:90,2] + 2.359;
   1:L PR[91] 10mm/sec CNT100;
   1:  PR[GP1:91,1] = PR[GP1:90,1] + 3.191;
   1:  PR[GP1:91,2] = PR[GP1:90,2] + 2.114;
   1:L PR[91] 10mm/sec CNT100;
   1:  PR[GP1:91,1] = PR[GP1:90,1] + 2.758;
   1:  PR[GP1:91,2] = PR[GP1:90,2] + 1.939;
   1:L PR[91] 10mm/sec CNT100;
   1:  PR[GP1:91,1] = PR[GP1:90,1] + 1.472;
   1:  PR[GP1:91,2] = PR[GP1:90,2] + 1.284;
   1:L PR[91] 10mm/sec CNT100;
   1:  PR[GP1:91,1] = PR[GP1:90,1] + -1.966;
   1:  PR[GP1:91,2] = PR[GP1:90,2] + 2.784;
   1:  PR[GP1:91,3] = PR[GP1:90,3] + 18.620;
   1:L PR[91] 10mm/sec CNT100;
   1:  PR[GP1:91,1] = PR[GP1:90,1] + -2.422;
   1:  PR[GP1:91,2] = PR[GP1:90,2] + 3.103;
   1:L PR[91] 10mm/sec CNT100;
   1:  PR[GP1:91,1] = PR[GP1:90,1] + -2.768;
   1:  PR[GP1:91,2] = PR[GP1:90,2] + 3.526;
   1:L PR[91] 10mm/sec CNT100;
   1:  PR[GP1:91,1] = PR[GP1:90,1] + -4.910;
   1:  PR[GP1:91,2] = PR[GP1:90,2] + 7.271;
   1:L PR[91] 10mm/sec CNT100;
   1:  PR[GP1:91,1] = PR[GP1:90,1] + -7.132;
   1:  PR[GP1:91,2] = PR[GP1:90,2] + 13.817;
   1:L PR[91] 10mm/sec CNT100;
   1:  PR[GP1:91,1] = PR[GP1:90,1] + -8.986;
   1:  PR[GP1:91,2] = PR[GP1:90,2] + 17.522;
   1:L PR[91] 10mm/sec CNT100;
   1:  PR[GP1:91,1] = PR[GP1:90,1] + -13.764;
   1:  PR[GP1:91,2] = PR[GP1:90,2] + 23.657;
   1:L PR[91] 10mm/sec CNT100;
   1:  PR[GP1:91,1] = PR[GP1:90,1] + -16.006;
   1:  PR[GP1:91,2] = PR[GP1:90,2] + 25.905;
   1:L PR[91] 10mm/sec CNT100;
   1:  PR[GP1:91,1] = PR[GP1:90,1] + -23.515;
   1:  PR[GP1:91,2] = PR[GP1:90,2] + 30.781;
   1:L PR[91] 10mm/sec CNT100;
   1:  PR[GP1:91,1] = PR[GP1:90,1] + -25.360;
   1:  PR[GP1:91,2] = PR[GP1:90,2] + 31.725;
   1:L PR[91] 10mm/sec CNT100;
   1:  PR[GP1:91,1] = PR[GP1:90,1] + -35.288;
   1:  PR[GP1:91,2] = PR[GP1:90,2] + 34.222;
   1:L PR[91] 10mm/sec CNT100;
   1:  PR[GP1:91,1] = PR[GP1:90,1] + -36.189;
   1:  PR[GP1:91,2] = PR[GP1:90,2] + 34.368;
   1:L PR[91] 10mm/sec CNT100;
   1:  PR[GP1:91,1] = PR[GP1:90,1] + -47.447;
   1:  PR[GP1:91,2] = PR[GP1:90,2] + 33.446;
   1:L PR[91] 10mm/sec CNT100;
   1:  PR[GP1:91,1] = PR[GP1:90,1] + -57.697;
   1:  PR[GP1:91,2] = PR[GP1:90,2] + 29.031;
   1:L PR[91] 10mm/sec CNT100;
   1:  PR[GP1:91,1] = PR[GP1:90,1] + -58.007;
   1:  PR[GP1:91,2] = PR[GP1:90,2] + 28.845;
   1:L PR[91] 10mm/sec CNT100;
   1:  PR[GP1:91,1] = PR[GP1:90,1] + -58.304;
   1:  PR[GP1:91,2] = PR[GP1:90,2] + 28.579;
   1:L PR[91] 10mm/sec CNT100;
   1:  PR[GP1:91,1] = PR[GP1:90,1] + -66.131;
   1:  PR[GP1:91,2] = PR[GP1:90,2] + 21.446;
   1:L PR[91] 10mm/sec CNT100;
   1:  PR[GP1:91,1] = PR[GP1:90,1] + -66.532;
   1:  PR[GP1:91,2] = PR[GP1:90,2] + 20.923;
   1:L PR[91] 10mm/sec CNT100;
   1:  PR[GP1:91,1] = PR[GP1:90,1] + -66.858;
   1:  PR[GP1:91,2] = PR[GP1:90,2] + 20.279;
   1:L PR[91] 10mm/sec CNT100;
   1:  PR[GP1:91,1] = PR[GP1:90,1] + -71.703;
   1:  PR[GP1:91,2] = PR[GP1:90,2] + 11.385;
   1:L PR[91] 10mm/sec CNT100;
   1:  PR[GP1:91,1] = PR[GP1:90,1] + -71.933;
   1:  PR[GP1:91,2] = PR[GP1:90,2] + 10.586;
   1:L PR[91] 10mm/sec CNT100;
   1:  PR[GP1:91,1] = PR[GP1:90,1] + -72.019;
   1:  PR[GP1:91,2] = PR[GP1:90,2] + 9.672;
   1:L PR[91] 10mm/sec CNT100;
   1:  PR[GP1:91,1] = PR[GP1:90,1] + -73.636;
   1:  PR[GP1:91,2] = PR[GP1:90,2] + -0.026;
   1:L PR[91] 10mm/sec CNT100;
   1:  PR[GP1:91,1] = PR[GP1:90,1] + -73.538;
   1:  PR[GP1:91,2] = PR[GP1:90,2] + -1.074;
   1:L PR[91] 10mm/sec CNT100;
   1:  PR[GP1:91,1] = PR[GP1:90,1] + -71.939;
   1:  PR[GP1:91,2] = PR[GP1:90,2] + -10.574;
   1:L PR[91] 10mm/sec CNT100;
   1:  PR[GP1:91,1] = PR[GP1:90,1] + -71.700;
   1:  PR[GP1:91,2] = PR[GP1:90,2] + -11.403;
   1:L PR[91] 10mm/sec CNT100;
   1:  PR[GP1:91,1] = PR[GP1:90,1] + -71.301;
   1:  PR[GP1:91,2] = PR[GP1:90,2] + -12.195;
   1:L PR[91] 10mm/sec CNT100;
   1:  PR[GP1:91,1] = PR[GP1:90,1] + -66.538;
   1:  PR[GP1:91,2] = PR[GP1:90,2] + -20.924;
   1:L PR[91] 10mm/sec CNT100;
   1:  PR[GP1:91,1] = PR[GP1:90,1] + -66.131;
   1:  PR[GP1:91,2] = PR[GP1:90,2] + -21.455;
   1:L PR[91] 10mm/sec CNT100;
   1:  PR[GP1:91,1] = PR[GP1:90,1] + -58.004;
   1:  PR[GP1:91,2] = PR[GP1:90,2] + -28.855;
   1:L PR[91] 10mm/sec CNT100;
   1:  PR[GP1:91,1] = PR[GP1:90,1] + -57.711;
   1:  PR[GP1:91,2] = PR[GP1:90,2] + -29.032;
   1:L PR[91] 10mm/sec CNT100;
   1:  PR[GP1:91,1] = PR[GP1:90,1] + -57.319;
   1:  PR[GP1:91,2] = PR[GP1:90,2] + -29.178;
   1:L PR[91] 10mm/sec CNT100;
   1:  PR[GP1:91,1] = PR[GP1:90,1] + -47.446;
   1:  PR[GP1:91,2] = PR[GP1:90,2] + -33.455;
   1:L PR[91] 10mm/sec CNT100;
   1:  PR[GP1:91,1] = PR[GP1:90,1] + -36.189;
   1:  PR[GP1:91,2] = PR[GP1:90,2] + -34.377;
   1:L PR[91] 10mm/sec CNT100;
   1:  PR[GP1:91,1] = PR[GP1:90,1] + -35.288;
   1:  PR[GP1:91,2] = PR[GP1:90,2] + -34.231;
   1:L PR[91] 10mm/sec CNT100;
   1:  PR[GP1:91,1] = PR[GP1:90,1] + -25.360;
   1:  PR[GP1:91,2] = PR[GP1:90,2] + -31.734;
   1:L PR[91] 10mm/sec CNT100;
   1:  PR[GP1:91,1] = PR[GP1:90,1] + -23.515;
   1:  PR[GP1:91,2] = PR[GP1:90,2] + -30.790;
   1:L PR[91] 10mm/sec CNT100;
   1:  PR[GP1:91,1] = PR[GP1:90,1] + -16.006;
   1:  PR[GP1:91,2] = PR[GP1:90,2] + -25.914;
   1:L PR[91] 10mm/sec CNT100;
   1:  PR[GP1:91,1] = PR[GP1:90,1] + -13.764;
   1:  PR[GP1:91,2] = PR[GP1:90,2] + -23.665;
   1:L PR[91] 10mm/sec CNT100;
   1:  PR[GP1:91,1] = PR[GP1:90,1] + -8.985;
   1:  PR[GP1:91,2] = PR[GP1:90,2] + -17.531;
   1:L PR[91] 10mm/sec CNT100;
   1:  PR[GP1:91,1] = PR[GP1:90,1] + -7.135;
   1:  PR[GP1:91,2] = PR[GP1:90,2] + -13.834;
   1:L PR[91] 10mm/sec CNT100;
   1:  PR[GP1:91,1] = PR[GP1:90,1] + -4.927;
   1:  PR[GP1:91,2] = PR[GP1:90,2] + -7.330;
   1:L PR[91] 10mm/sec CNT100;
   1:  PR[GP1:91,1] = PR[GP1:90,1] + -4.158;
   1:  PR[GP1:91,2] = PR[GP1:90,2] + -5.166;
   1:L PR[91] 10mm/sec CNT100;
   1:  PR[GP1:91,1] = PR[GP1:90,1] + -2.386;
   1:  PR[GP1:91,2] = PR[GP1:90,2] + -3.206;
   1:L PR[91] 10mm/sec CNT100;
   1:  PR[GP1:91,1] = PR[GP1:90,1] + -1.862;
   1:  PR[GP1:91,2] = PR[GP1:90,2] + -2.886;
   1:L PR[91] 10mm/sec CNT100;
   1:  PR[GP1:91,1] = PR[GP1:90,1] + -1.524;
   1:  PR[GP1:91,2] = PR[GP1:90,2] + -2.483;
   1:L PR[91] 10mm/sec CNT100;
   1:  PR[GP1:91,1] = PR[GP1:90,1] + 2.533;
   1:  PR[GP1:91,2] = PR[GP1:90,2] + -2.795;
   1:L PR[91] 10mm/sec CNT100;
   1:  PR[GP1:91,1] = PR[GP1:90,1] + 2.729;
   1:  PR[GP1:91,2] = PR[GP1:90,2] + -2.954;
   1:L PR[91] 10mm/sec CNT100;
   1:  PR[GP1:91,1] = PR[GP1:90,1] + 3.184;
   1:  PR[GP1:91,2] = PR[GP1:90,2] + -2.949;
   1:L PR[91] 10mm/sec CNT100;
   1:  PR[GP1:91,1] = PR[GP1:90,1] + 5.000;
   1:  PR[GP1:91,2] = PR[GP1:90,2] + -6.404;
   1:L PR[91] 10mm/sec CNT100;
   1:  PR[GP1:91,1] = PR[GP1:90,1] + 5.709;
   1:  PR[GP1:91,2] = PR[GP1:90,2] + -7.222;
   1:L PR[91] 10mm/sec CNT100;
   1:  PR[GP1:91,1] = PR[GP1:90,1] + 7.952;
   1:  PR[GP1:91,2] = PR[GP1:90,2] + -13.829;
   1:L PR[91] 10mm/sec CNT100;
   1:  PR[GP1:91,1] = PR[GP1:90,1] + 9.802;
   1:  PR[GP1:91,2] = PR[GP1:90,2] + -17.519;
   1:L PR[91] 10mm/sec CNT100;
   1:  PR[GP1:91,1] = PR[GP1:90,1] + 14.580;
   1:  PR[GP1:91,2] = PR[GP1:90,2] + -23.657;
   1:L PR[91] 10mm/sec CNT100;
   1:  PR[GP1:91,1] = PR[GP1:90,1] + 16.822;
   1:  PR[GP1:91,2] = PR[GP1:90,2] + -25.912;
   1:L PR[91] 10mm/sec CNT100;
   1:  PR[GP1:91,1] = PR[GP1:90,1] + 24.331;
   1:  PR[GP1:91,2] = PR[GP1:90,2] + -30.788;
   1:L PR[91] 10mm/sec CNT100;
   1:  PR[GP1:91,1] = PR[GP1:90,1] + 26.177;
   1:  PR[GP1:91,2] = PR[GP1:90,2] + -31.732;
   1:L PR[91] 10mm/sec CNT100;
   1:  PR[GP1:91,1] = PR[GP1:90,1] + 36.105;
   1:  PR[GP1:91,2] = PR[GP1:90,2] + -34.230;
   1:L PR[91] 10mm/sec CNT100;
   1:  PR[GP1:91,1] = PR[GP1:90,1] + 37.007;
   1:  PR[GP1:91,2] = PR[GP1:90,2] + -34.377;
   1:L PR[91] 10mm/sec CNT100;
   1:  PR[GP1:91,1] = PR[GP1:90,1] + 48.246;
   1:  PR[GP1:91,2] = PR[GP1:90,2] + -33.458;
   1:L PR[91] 10mm/sec CNT100;
   1:  PR[GP1:91,1] = PR[GP1:90,1] + 58.517;
   1:  PR[GP1:91,2] = PR[GP1:90,2] + -29.041;
   1:L PR[91] 10mm/sec CNT100;
   1:  PR[GP1:91,1] = PR[GP1:90,1] + 58.824;
   1:  PR[GP1:91,2] = PR[GP1:90,2] + -28.856;
   1:L PR[91] 10mm/sec CNT100;
   1:  PR[GP1:91,1] = PR[GP1:90,1] + 66.951;
   1:  PR[GP1:91,2] = PR[GP1:90,2] + -21.454;
   1:L PR[91] 10mm/sec CNT100;
   1:  PR[GP1:91,1] = PR[GP1:90,1] + 67.353;
   1:  PR[GP1:91,2] = PR[GP1:90,2] + -20.931;
   1:L PR[91] 10mm/sec CNT100;
   1:  PR[GP1:91,1] = PR[GP1:90,1] + 67.678;
   1:  PR[GP1:91,2] = PR[GP1:90,2] + -20.286;
   1:L PR[91] 10mm/sec CNT100;
   1:  PR[GP1:91,1] = PR[GP1:90,1] + 72.524;
   1:  PR[GP1:91,2] = PR[GP1:90,2] + -11.398;
   1:L PR[91] 10mm/sec CNT100;
   1:  PR[GP1:91,1] = PR[GP1:90,1] + 72.754;
   1:  PR[GP1:91,2] = PR[GP1:90,2] + -10.599;
   1:L PR[91] 10mm/sec CNT100;
   1:  PR[GP1:91,1] = PR[GP1:90,1] + 72.839;
   1:  PR[GP1:91,2] = PR[GP1:90,2] + -9.685;
   1:L PR[91] 10mm/sec CNT100;
   1:  PR[GP1:91,1] = PR[GP1:90,1] + 74.457;
   1:  PR[GP1:91,2] = PR[GP1:90,2] + 0.017;
   1:L PR[91] 10mm/sec CNT100;
   1:  PR[GP1:91,1] = PR[GP1:90,1] + 74.359;
   1:  PR[GP1:91,2] = PR[GP1:90,2] + 1.066;
   1:L PR[91] 10mm/sec CNT100;
   1:  PR[GP1:91,1] = PR[GP1:90,1] + 72.760;
   1:  PR[GP1:91,2] = PR[GP1:90,2] + 10.569;
   1:L PR[91] 10mm/sec CNT100;
   1:  PR[GP1:91,1] = PR[GP1:90,1] + 72.521;
   1:  PR[GP1:91,2] = PR[GP1:90,2] + 11.398;
   1:L PR[91] 10mm/sec CNT100;
   1:  PR[GP1:91,1] = PR[GP1:90,1] + 72.121;
   1:  PR[GP1:91,2] = PR[GP1:90,2] + 12.190;
   1:L PR[91] 10mm/sec CNT100;
   1:  PR[GP1:91,1] = PR[GP1:90,1] + 67.359;
   1:  PR[GP1:91,2] = PR[GP1:90,2] + 20.914;
   1:L PR[91] 10mm/sec CNT100;
   1:  PR[GP1:91,1] = PR[GP1:90,1] + 66.951;
   1:  PR[GP1:91,2] = PR[GP1:90,2] + 21.445;
   1:L PR[91] 10mm/sec CNT100;
   1:  PR[GP1:91,1] = PR[GP1:90,1] + 58.824;
   1:  PR[GP1:91,2] = PR[GP1:90,2] + 28.848;
   1:L PR[91] 10mm/sec CNT100;
   1:  PR[GP1:91,1] = PR[GP1:90,1] + 58.530;
   1:  PR[GP1:91,2] = PR[GP1:90,2] + 29.025;
   1:L PR[91] 10mm/sec CNT100;
   1:  PR[GP1:91,1] = PR[GP1:90,1] + 58.139;
   1:  PR[GP1:91,2] = PR[GP1:90,2] + 29.170;
   1:L PR[91] 10mm/sec CNT100;
   1:  PR[GP1:91,1] = PR[GP1:90,1] + 48.265;
   1:  PR[GP1:91,2] = PR[GP1:90,2] + 33.446;
   1:L PR[91] 10mm/sec CNT100;
   1:  PR[GP1:91,1] = PR[GP1:90,1] + 37.007;
   1:  PR[GP1:91,2] = PR[GP1:90,2] + 34.368;
   1:L PR[91] 10mm/sec CNT100;
   1:  PR[GP1:91,1] = PR[GP1:90,1] + 36.105;
   1:  PR[GP1:91,2] = PR[GP1:90,2] + 34.221;
   1:L PR[91] 10mm/sec CNT100;
   1:  PR[GP1:91,1] = PR[GP1:90,1] + 26.177;
   1:  PR[GP1:91,2] = PR[GP1:90,2] + 31.723;
   1:L PR[91] 10mm/sec CNT100;
   1:  PR[GP1:91,1] = PR[GP1:90,1] + 24.331;
   1:  PR[GP1:91,2] = PR[GP1:90,2] + 30.779;
   1:L PR[91] 10mm/sec CNT100;
   1:  PR[GP1:91,1] = PR[GP1:90,1] + 16.822;
   1:  PR[GP1:91,2] = PR[GP1:90,2] + 25.903;
   1:L PR[91] 10mm/sec CNT100;
   1:  PR[GP1:91,1] = PR[GP1:90,1] + 14.580;
   1:  PR[GP1:91,2] = PR[GP1:90,2] + 23.648;
   1:L PR[91] 10mm/sec CNT100;
   1:  PR[GP1:91,1] = PR[GP1:90,1] + 9.802;
   1:  PR[GP1:91,2] = PR[GP1:90,2] + 17.510;
   1:L PR[91] 10mm/sec CNT100;
   1:  PR[GP1:91,1] = PR[GP1:90,1] + 7.949;
   1:  PR[GP1:91,2] = PR[GP1:90,2] + 13.812;
   1:L PR[91] 10mm/sec CNT100;
   1:  PR[GP1:91,1] = PR[GP1:90,1] + 5.745;
   1:  PR[GP1:91,2] = PR[GP1:90,2] + 7.321;
   1:L PR[91] 10mm/sec CNT100;
   1:  PR[GP1:91,1] = PR[GP1:90,1] + 4.980;
   1:  PR[GP1:91,2] = PR[GP1:90,2] + 5.164;
   1:L PR[91] 10mm/sec CNT100;
   1:  PR[GP1:91,1] = PR[GP1:90,1] + 4.460;
   1:  PR[GP1:91,2] = PR[GP1:90,2] + 4.534;
   1:L PR[91] 10mm/sec CNT100;
   1:  PR[GP1:91,1] = PR[GP1:90,1] + 2.948;
   1:  PR[GP1:91,2] = PR[GP1:90,2] + 2.889;
   1:L PR[91] 10mm/sec CNT100;
   1:  PR[GP1:91,1] = PR[GP1:90,1] + 2.230;
   1:  PR[GP1:91,2] = PR[GP1:90,2] + 2.492;
   1:L PR[91] 10mm/sec CNT100;
   1:  PR[GP1:91,1] = PR[GP1:90,1] + 1.833;
   1:  PR[GP1:91,2] = PR[GP1:90,2] + 2.496;
   1:L PR[91] 10mm/sec CNT100;
   1:  PR[GP1:91,1] = PR[GP1:90,1] + 1.358;
   1:  PR[GP1:91,2] = PR[GP1:90,2] + 3.658;
   1:  PR[GP1:91,3] = PR[GP1:90,3] + 19.950;
   1:L PR[91] 10mm/sec CNT100;
   1:  PR[GP1:91,1] = PR[GP1:90,1] + -1.916;
   1:  PR[GP1:91,2] = PR[GP1:90,2] + 3.906;
   1:L PR[91] 10mm/sec CNT100;
   1:  PR[GP1:91,1] = PR[GP1:90,1] + -2.335;
   1:  PR[GP1:91,2] = PR[GP1:90,2] + 4.200;
   1:L PR[91] 10mm/sec CNT100;
   1:  PR[GP1:91,1] = PR[GP1:90,1] + -3.086;
   1:  PR[GP1:91,2] = PR[GP1:90,2] + 5.120;
   1:L PR[91] 10mm/sec CNT100;
   1:  PR[GP1:91,1] = PR[GP1:90,1] + -4.857;
   1:  PR[GP1:91,2] = PR[GP1:90,2] + 8.231;
   1:L PR[91] 10mm/sec CNT100;
   1:  PR[GP1:91,1] = PR[GP1:90,1] + -6.352;
   1:  PR[GP1:91,2] = PR[GP1:90,2] + 12.633;
   1:L PR[91] 10mm/sec CNT100;
   1:  PR[GP1:91,1] = PR[GP1:90,1] + -9.159;
   1:  PR[GP1:91,2] = PR[GP1:90,2] + 18.245;
   1:L PR[91] 10mm/sec CNT100;
   1:  PR[GP1:91,1] = PR[GP1:90,1] + -12.624;
   1:  PR[GP1:91,2] = PR[GP1:90,2] + 22.694;
   1:L PR[91] 10mm/sec CNT100;
   1:  PR[GP1:91,1] = PR[GP1:90,1] + -16.284;
   1:  PR[GP1:91,2] = PR[GP1:90,2] + 26.365;
   1:L PR[91] 10mm/sec CNT100;
   1:  PR[GP1:91,1] = PR[GP1:90,1] + -22.097;
   1:  PR[GP1:91,2] = PR[GP1:90,2] + 30.140;
   1:L PR[91] 10mm/sec CNT100;
   1:  PR[GP1:91,1] = PR[GP1:90,1] + -25.642;
   1:  PR[GP1:91,2] = PR[GP1:90,2] + 31.952;
   1:L PR[91] 10mm/sec CNT100;
   1:  PR[GP1:91,1] = PR[GP1:90,1] + -33.739;
   1:  PR[GP1:91,2] = PR[GP1:90,2] + 33.989;
   1:L PR[91] 10mm/sec CNT100;
   1:  PR[GP1:91,1] = PR[GP1:90,1] + -36.406;
   1:  PR[GP1:91,2] = PR[GP1:90,2] + 34.421;
   1:L PR[91] 10mm/sec CNT100;
   1:  PR[GP1:91,1] = PR[GP1:90,1] + -46.034;
   1:  PR[GP1:91,2] = PR[GP1:90,2] + 33.632;
   1:L PR[91] 10mm/sec CNT100;
   1:  PR[GP1:91,1] = PR[GP1:90,1] + -47.540;
   1:  PR[GP1:91,2] = PR[GP1:90,2] + 33.403;
   1:L PR[91] 10mm/sec CNT100;
   1:  PR[GP1:91,1] = PR[GP1:90,1] + -57.367;
   1:  PR[GP1:91,2] = PR[GP1:90,2] + 29.131;
   1:L PR[91] 10mm/sec CNT100;
   1:  PR[GP1:91,1] = PR[GP1:90,1] + -57.878;
   1:  PR[GP1:91,2] = PR[GP1:90,2] + 28.876;
   1:L PR[91] 10mm/sec CNT100;
   1:  PR[GP1:91,1] = PR[GP1:90,1] + -66.272;
   1:  PR[GP1:91,2] = PR[GP1:90,2] + 21.219;
   1:L PR[91] 10mm/sec CNT100;
   1:  PR[GP1:91,1] = PR[GP1:90,1] + -71.715;
   1:  PR[GP1:91,2] = PR[GP1:90,2] + 11.229;
   1:L PR[91] 10mm/sec CNT100;
   1:  PR[GP1:91,1] = PR[GP1:90,1] + -71.739;
   1:  PR[GP1:91,2] = PR[GP1:90,2] + 11.147;
   1:L PR[91] 10mm/sec CNT100;
   1:  PR[GP1:91,1] = PR[GP1:90,1] + -71.755;
   1:  PR[GP1:91,2] = PR[GP1:90,2] + 10.975;
   1:L PR[91] 10mm/sec CNT100;
   1:  PR[GP1:91,1] = PR[GP1:90,1] + -73.590;
   1:  PR[GP1:91,2] = PR[GP1:90,2] + -0.026;
   1:L PR[91] 10mm/sec CNT100;
   1:  PR[GP1:91,1] = PR[GP1:90,1] + -73.559;
   1:  PR[GP1:91,2] = PR[GP1:90,2] + -0.359;
   1:L PR[91] 10mm/sec CNT100;
   1:  PR[GP1:91,1] = PR[GP1:90,1] + -71.745;
   1:  PR[GP1:91,2] = PR[GP1:90,2] + -11.134;
   1:L PR[91] 10mm/sec CNT100;
   1:  PR[GP1:91,1] = PR[GP1:90,1] + -71.712;
   1:  PR[GP1:91,2] = PR[GP1:90,2] + -11.247;
   1:L PR[91] 10mm/sec CNT100;
   1:  PR[GP1:91,1] = PR[GP1:90,1] + -71.648;
   1:  PR[GP1:91,2] = PR[GP1:90,2] + -11.374;
   1:L PR[91] 10mm/sec CNT100;
   1:  PR[GP1:91,1] = PR[GP1:90,1] + -66.271;
   1:  PR[GP1:91,2] = PR[GP1:90,2] + -21.230;
   1:L PR[91] 10mm/sec CNT100;
   1:  PR[GP1:91,1] = PR[GP1:90,1] + -57.878;
   1:  PR[GP1:91,2] = PR[GP1:90,2] + -28.885;
   1:L PR[91] 10mm/sec CNT100;
   1:  PR[GP1:91,1] = PR[GP1:90,1] + -57.367;
   1:  PR[GP1:91,2] = PR[GP1:90,2] + -29.140;
   1:L PR[91] 10mm/sec CNT100;
   1:  PR[GP1:91,1] = PR[GP1:90,1] + -47.540;
   1:  PR[GP1:91,2] = PR[GP1:90,2] + -33.412;
   1:L PR[91] 10mm/sec CNT100;
   1:  PR[GP1:91,1] = PR[GP1:90,1] + -46.034;
   1:  PR[GP1:91,2] = PR[GP1:90,2] + -33.640;
   1:L PR[91] 10mm/sec CNT100;
   1:  PR[GP1:91,1] = PR[GP1:90,1] + -36.406;
   1:  PR[GP1:91,2] = PR[GP1:90,2] + -34.430;
   1:L PR[91] 10mm/sec CNT100;
   1:  PR[GP1:91,1] = PR[GP1:90,1] + -33.739;
   1:  PR[GP1:91,2] = PR[GP1:90,2] + -33.998;
   1:L PR[91] 10mm/sec CNT100;
   1:  PR[GP1:91,1] = PR[GP1:90,1] + -25.642;
   1:  PR[GP1:91,2] = PR[GP1:90,2] + -31.961;
   1:L PR[91] 10mm/sec CNT100;
   1:  PR[GP1:91,1] = PR[GP1:90,1] + -22.097;
   1:  PR[GP1:91,2] = PR[GP1:90,2] + -30.149;
   1:L PR[91] 10mm/sec CNT100;
   1:  PR[GP1:91,1] = PR[GP1:90,1] + -16.284;
   1:  PR[GP1:91,2] = PR[GP1:90,2] + -26.374;
   1:L PR[91] 10mm/sec CNT100;
   1:  PR[GP1:91,1] = PR[GP1:90,1] + -12.624;
   1:  PR[GP1:91,2] = PR[GP1:90,2] + -22.703;
   1:L PR[91] 10mm/sec CNT100;
   1:  PR[GP1:91,1] = PR[GP1:90,1] + -9.159;
   1:  PR[GP1:91,2] = PR[GP1:90,2] + -18.254;
   1:L PR[91] 10mm/sec CNT100;
   1:  PR[GP1:91,1] = PR[GP1:90,1] + -6.356;
   1:  PR[GP1:91,2] = PR[GP1:90,2] + -12.654;
   1:L PR[91] 10mm/sec CNT100;
   1:  PR[GP1:91,1] = PR[GP1:90,1] + -4.874;
   1:  PR[GP1:91,2] = PR[GP1:90,2] + -8.290;
   1:L PR[91] 10mm/sec CNT100;
   1:  PR[GP1:91,1] = PR[GP1:90,1] + -4.232;
   1:  PR[GP1:91,2] = PR[GP1:90,2] + -6.475;
   1:L PR[91] 10mm/sec CNT100;
   1:  PR[GP1:91,1] = PR[GP1:90,1] + -2.758;
   1:  PR[GP1:91,2] = PR[GP1:90,2] + -4.845;
   1:L PR[91] 10mm/sec CNT100;
   1:  PR[GP1:91,1] = PR[GP1:90,1] + -2.332;
   1:  PR[GP1:91,2] = PR[GP1:90,2] + -4.585;
   1:L PR[91] 10mm/sec CNT100;
   1:  PR[GP1:91,1] = PR[GP1:90,1] + -1.546;
   1:  PR[GP1:91,2] = PR[GP1:90,2] + -3.645;
   1:L PR[91] 10mm/sec CNT100;
   1:  PR[GP1:91,1] = PR[GP1:90,1] + 1.994;
   1:  PR[GP1:91,2] = PR[GP1:90,2] + -3.917;
   1:L PR[91] 10mm/sec CNT100;
   1:  PR[GP1:91,1] = PR[GP1:90,1] + 2.158;
   1:  PR[GP1:91,2] = PR[GP1:90,2] + -4.050;
   1:L PR[91] 10mm/sec CNT100;
   1:  PR[GP1:91,1] = PR[GP1:90,1] + 3.087;
   1:  PR[GP1:91,2] = PR[GP1:90,2] + -4.041;
   1:L PR[91] 10mm/sec CNT100;
   1:  PR[GP1:91,1] = PR[GP1:90,1] + 4.659;
   1:  PR[GP1:91,2] = PR[GP1:90,2] + -7.034;
   1:L PR[91] 10mm/sec CNT100;
   1:  PR[GP1:91,1] = PR[GP1:90,1] + 5.655;
   1:  PR[GP1:91,2] = PR[GP1:90,2] + -8.181;
   1:L PR[91] 10mm/sec CNT100;
